  LIN {X -999.998,Y -0.298,Z -43.502,A -90.00011,B 0.00000,C -180.00000} ; release
  LIN {X -999.998,Y -0.298,Z 256.498,A -90.00011,B 0.00000,C -180.00000} ; retreat
  ; Step 2683, bar 145
  LIN {X -874.998,Y -0.298,Z 1164.733,A -90.00011,B 0.00000,C -180.00000} ; outside
  LIN {X -874.998,Y -0.298,Z 206.498,A -90.00011,B 0.00000,C -180.00000} ; preinsert
  LIN {X -874.998,Y -0.298,Z -43.502,A -90.00011,B 0.00000,C -180.00000} ; insert
  LIN {X -874.998,Y -0.298,Z -43.502,A -90.00011,B 0.00000,C -180.00000} ; release
  LIN {X -874.998,Y -0.298,Z 256.498,A -90.00011,B 0.00000,C -180.00000} ; retreat
  ; Step 2684, bar 144
  LIN {X -749.998,Y -0.298,Z 1164.733,A -90.00011,B 0.00000,C -180.00000} ; outside
  LIN {X -749.998,Y -0.298,Z 206.498,A -90.00011,B 0.00000,C -180.00000} ; preinsert
  LIN {X -749.998,Y -0.298,Z -43.502,A -90.00011,B 0.00000,C -180.00000} ; insert
  LIN {X -749.998,Y -0.298,Z -43.502,A -90.00011,B 0.00000,C -180.00000} ; release
  LIN {X -749.998,Y -0.298,Z 256.498,A -90.00011,B 0.00000,C -180.00000} ; retreat
  ; Step 2685, bar 143
  LIN {X -624.998,Y -0.298,Z 1164.733,A -90.00011,B 0.00000,C -180.00000} ; outside
  LIN {X -624.998,Y -0.298,Z 206.498,A -90.00011,B 0.00000,C -180.00000} ; preinsert
  LIN {X -624.998,Y -0.298,Z -43.502,A -90.00011,B 0.00000,C -180.00000} ; insert
  LIN {X -624.998,Y -0.298,Z -43.502,A -90.00011,B 0.00000,C -180.00000} ; release
  LIN {X -624.998,Y -0.298,Z 256.498,A -90.00011,B 0.00000,C -180.00000} ; retreat
  ; Step 2686, bar 142
  LIN {X -499.998,Y -0.298,Z 1164.733,A -90.00011,B 0.00000,C -180.00000} ; outside
  LIN {X -499.998,Y -0.298,Z 206.498,A -90.00011,B 0.00000,C -180.00000} ; preinsert
  LIN {X -499.998,Y -0.298,Z -43.502,A -90.00011,B 0.00000,C -180.00000} ; insert
  LIN {X -499.998,Y -0.298,Z -43.502,A -90.00011,B 0.00000,C -180.00000} ; release
  LIN {X -499.998,Y -0.298,Z 256.498,A -90.00011,B 0.00000,C -180.00000} ; retreat
  ; Step 2687, bar 141
  LIN {X -374.998,Y -0.298,Z 1164.733,A -90.00011,B 0.00000,C -180.00000} ; outside
  LIN {X -374.998,Y -0.298,Z 206.498,A -90.00011,B 0.00000,C -180.00000} ; preinsert
  LIN {X -374.998,Y -0.298,Z -43.502,A -90.00011,B 0.00000,C -180.00000} ; insert
  LIN {X -374.998,Y -0.298,Z -43.502,A -90.00011,B 0.00000,C -180.00000} ; release
  LIN {X -374.998,Y -0.298,Z 256.498,A -90.00011,B 0.00000,C -180.00000} ; retreat
  ; Step 2688, bar 140
  LIN {X -249.998,Y -0.298,Z 1164.733,A -90.00011,B 0.00000,C -180.00000} ; outside
  LIN {X -249.998,Y -0.298,Z 206.498,A -90.00011,B 0.00000,C -180.00000} ; preinsert
  LIN {X -249.998,Y -0.298,Z -43.502,A -90.00011,B 0.00000,C -180.00000} ; insert
  LIN {X -249.998,Y -0.298,Z -43.502,A -90.00011,B 0.00000,C -180.00000} ; release
  LIN {X -249.998,Y -0.298,Z 256.498,A -90.00011,B 0.00000,C -180.00000} ; retreat
  ; Step 2689, bar 139
  LIN {X -124.998,Y -0.298,Z 1164.733,A -90.00011,B 0.00000,C -180.00000} ; outside
  LIN {X -124.998,Y -0.298,Z 206.498,A -90.00011,B 0.00000,C -180.00000} ; preinsert
  LIN {X -124.998,Y -0.298,Z -43.502,A -90.00011,B 0.00000,C -180.00000} ; insert
  LIN {X -124.998,Y -0.298,Z -43.502,A -90.00011,B 0.00000,C -180.00000} ; release
  LIN {X -124.998,Y -0.298,Z 256.498,A -90.00011,B 0.00000,C -180.00000} ; retreat
  ; Step 2690, bar 0
  LIN {X -0.034,Y -0.300,Z 1164.951,A -90.01312,B 0.00000,C -180.00000} ; outside
  LIN {X -0.034,Y -0.300,Z 206.586,A -90.01312,B 0.00000,C -180.00000} ; preinsert
  LIN {X -0.034,Y -0.300,Z -43.414,A -90.01312,B 0.00000,C -180.00000} ; insert
  LIN {X -0.034,Y -0.300,Z -43.414,A -90.01312,B 0.00000,C -180.00000} ; release
  LIN {X -0.034,Y -0.300,Z 256.586,A -90.01312,B 0.00000,C -180.00000} ; retreat
  ; Step 2691, bar 1
  LIN {X 124.966,Y -0.300,Z 1164.951,A -90.01312,B 0.00000,C -180.00000} ; outside
  LIN {X 124.966,Y -0.300,Z 206.586,A -90.01312,B 0.00000,C -180.00000} ; preinsert
  LIN {X 124.966,Y -0.300,Z -43.414,A -90.01312,B 0.00000,C -180.00000} ; insert
  LIN {X 124.966,Y -0.300,Z -43.414,A -90.01312,B 0.00000,C -180.00000} ; release
  LIN {X 124.966,Y -0.300,Z 256.586,A -90.01312,B 0.00000,C -180.00000} ; retreat
  ; Step 2692, bar 2
  LIN {X 249.966,Y -0.300,Z 1164.951,A -90.01312,B 0.00000,C -180.00000} ; outside
  LIN {X 249.966,Y -0.300,Z 206.586,A -90.01312,B 0.00000,C -180.00000} ; preinsert
  LIN {X 249.966,Y -0.300,Z -43.414,A -90.01312,B 0.00000,C -180.00000} ; insert
  LIN {X 249.966,Y -0.300,Z -43.414,A -90.01312,B 0.00000,C -180.00000} ; release
  LIN {X 249.966,Y -0.300,Z 256.586,A -90.01312,B 0.00000,C -180.00000} ; retreat
  ; Step 2693, bar 3
  LIN {X 374.966,Y -0.300,Z 1164.951,A -90.01312,B 0.00000,C -180.00000} ; outside
  LIN {X 374.966,Y -0.300,Z 206.586,A -90.01312,B 0.00000,C -180.00000} ; preinsert
  LIN {X 374.966,Y -0.300,Z -43.414,A -90.01312,B 0.00000,C -180.00000} ; insert
  LIN {X 374.966,Y -0.300,Z -43.414,A -90.01312,B 0.00000,C -180.00000} ; release
  LIN {X 374.966,Y -0.300,Z 256.586,A -90.01312,B 0.00000,C -180.00000} ; retreat
  ; Step 2694, bar 4
  LIN {X 499.966,Y -0.300,Z 1164.951,A -90.01312,B 0.00000,C -180.00000} ; outside
  LIN {X 499.966,Y -0.300,Z 206.586,A -90.01312,B 0.00000,C -180.00000} ; preinsert
  LIN {X 499.966,Y -0.300,Z -43.414,A -90.01312,B 0.00000,C -180.00000} ; insert
  LIN {X 499.966,Y -0.300,Z -43.414,A -90.01312,B 0.00000,C -180.00000} ; release
  LIN {X 499.966,Y -0.300,Z 256.586,A -90.01312,B 0.00000,C -180.00000} ; retreat
  ; Step 2695, bar 5
  LIN {X 624.966,Y -0.300,Z 1164.951,A -90.01312,B 0.00000,C -180.00000} ; outside
  LIN {X 624.966,Y -0.300,Z 206.586,A -90.01312,B 0.00000,C -180.00000} ; preinsert
  LIN {X 624.966,Y -0.300,Z -43.414,A -90.01312,B 0.00000,C -180.00000} ; insert
  LIN {X 624.966,Y -0.300,Z -43.414,A -90.01312,B 0.00000,C -180.00000} ; release
  LIN {X 624.966,Y -0.300,Z 256.586,A -90.01312,B 0.00000,C -180.00000} ; retreat
  ; Step 2696, bar 6
  LIN {X 749.966,Y -0.300,Z 1164.951,A -90.01312,B 0.00000,C -180.00000} ; outside
  LIN {X 749.966,Y -0.300,Z 206.586,A -90.01312,B 0.00000,C -180.00000} ; preinsert
  LIN {X 749.966,Y -0.300,Z -43.414,A -90.01312,B 0.00000,C -180.00000} ; insert
  LIN {X 749.966,Y -0.300,Z -43.414,A -90.01312,B 0.00000,C -180.00000} ; release
  LIN {X 749.966,Y -0.300,Z 256.586,A -90.01312,B 0.00000,C -180.00000} ; retreat
  ; Step 2697, bar 7
  LIN {X 874.966,Y -0.300,Z 1164.951,A -90.01312,B 0.00000,C -180.00000} ; outside
  LIN {X 874.966,Y -0.300,Z 206.586,A -90.01312,B 0.00000,C -180.00000} ; preinsert
  LIN {X 874.966,Y -0.300,Z -43.414,A -90.01312,B 0.00000,C -180.00000} ; insert
  LIN {X 874.966,Y -0.300,Z -43.414,A -90.01312,B 0.00000,C -180.00000} ; release
  LIN {X 874.966,Y -0.300,Z 256.586,A -90.01312,B 0.00000,C -180.00000} ; retreat
  ; Step 2698, bar 8
  LIN {X 999.966,Y -0.300,Z 1164.951,A -90.01312,B 0.00000,C -180.00000} ; outside
  LIN {X 999.966,Y -0.300,Z 206.586,A -90.01312,B 0.00000,C -180.00000} ; preinsert
  LIN {X 999.966,Y -0.300,Z -43.414,A -90.01312,B 0.00000,C -180.00000} ; insert
  LIN {X 999.966,Y -0.300,Z -43.414,A -90.01312,B 0.00000,C -180.00000} ; release
  LIN {X 999.966,Y -0.300,Z 256.586,A -90.01312,B 0.00000,C -180.00000} ; retreat
  ; Step 2699, bar 9
  LIN {X 1124.966,Y -0.300,Z 1164.951,A -90.01312,B 0.00000,C -180.00000} ; outside
  LIN {X 1124.966,Y -0.300,Z 206.586,A -90.01312,B 0.00000,C -180.00000} ; preinsert
  LIN {X 1124.966,Y -0.300,Z -43.414,A -90.01312,B 0.00000,C -180.00000} ; insert
  LIN {X 1124.966,Y -0.300,Z -43.414,A -90.01312,B 0.00000,C -180.00000} ; release
  LIN {X 1124.966,Y -0.300,Z 256.586,A -90.01312,B 0.00000,C -180.00000} ; retreat
  ; Step 2700, bar 10
  LIN {X 1249.966,Y -0.300,Z 1164.951,A -90.01312,B 0.00000,C -180.00000} ; outside
  LIN {X 1249.966,Y -0.300,Z 206.586,A -90.01312,B 0.00000,C -180.00000} ; preinsert
  LIN {X 1249.966,Y -0.300,Z -43.414,A -90.01312,B 0.00000,C -180.00000} ; insert
  LIN {X 1249.966,Y -0.300,Z -43.414,A -90.01312,B 0.00000,C -180.00000} ; release
  LIN {X 1249.966,Y -0.300,Z 256.586,A -90.01312,B 0.00000,C -180.00000} ; retreat
  ; Step 2701, bar 11
  LIN {X 1374.966,Y -0.300,Z 1164.951,A -90.01312,B 0.00000,C -180.00000} ; outside
  LIN {X 1374.966,Y -0.300,Z 206.586,A -90.01312,B 0.00000,C -180.00000} ; preinsert
  LIN {X 1374.966,Y -0.300,Z -43.414,A -90.01312,B 0.00000,C -180.00000} ; insert
  LIN {X 1374.966,Y -0.300,Z -43.414,A -90.01312,B 0.00000,C -180.00000} ; release
  LIN {X 1374.966,Y -0.300,Z 256.586,A -90.01312,B 0.00000,C -180.00000} ; retreat
  ; Step 2702, bar 12
  LIN {X 1499.966,Y -0.300,Z 1164.951,A -90.01312,B 0.00000,C -180.00000} ; outside
  LIN {X 1499.966,Y -0.300,Z 206.586,A -90.01312,B 0.00000,C -180.00000} ; preinsert
  LIN {X 1499.966,Y -0.300,Z -43.414,A -90.01312,B 0.00000,C -180.00000} ; insert
  LIN {X 1499.966,Y -0.300,Z -43.414,A -90.01312,B 0.00000,C -180.00000} ; release
  LIN {X 1499.966,Y -0.300,Z 256.586,A -90.01312,B 0.00000,C -180.00000} ; retreat
  ; Step 2703, bar 13
  LIN {X 1624.966,Y -0.300,Z 1164.951,A -90.01312,B 0.00000,C -180.00000} ; outside
  LIN {X 1624.966,Y -0.300,Z 206.586,A -90.01312,B 0.00000,C -180.00000} ; preinsert
  LIN {X 1624.966,Y -0.300,Z -43.414,A -90.01312,B 0.00000,C -180.00000} ; insert
  LIN {X 1624.966,Y -0.300,Z -43.414,A -90.01312,B 0.00000,C -180.00000} ; release
  LIN {X 1624.966,Y -0.300,Z 256.586,A -90.01312,B 0.00000,C -180.00000} ; retreat
  ; Step 2704, bar 14
  LIN {X 1749.966,Y -0.300,Z 1164.951,A -90.01312,B 0.00000,C -180.00000} ; outside
  LIN {X 1749.966,Y -0.300,Z 206.586,A -90.01312,B 0.00000,C -180.00000} ; preinsert
  LIN {X 1749.966,Y -0.300,Z -43.414,A -90.01312,B 0.00000,C -180.00000} ; insert
  LIN {X 1749.966,Y -0.300,Z -43.414,A -90.01312,B 0.00000,C -180.00000} ; release
  LIN {X 1749.966,Y -0.300,Z 256.586,A -90.01312,B 0.00000,C -180.00000} ; retreat
  ; Step 2705, bar 16
  LIN {X 1874.966,Y -0.300,Z 1164.951,A -90.01312,B 0.00000,C -180.00000} ; outside
  LIN {X 1874.966,Y -0.300,Z 206.586,A -90.01312,B 0.00000,C -180.00000} ; preinsert
  LIN {X 1874.966,Y -0.300,Z -43.414,A -90.01312,B 0.00000,C -180.00000} ; insert
  LIN {X 1874.966,Y -0.300,Z -43.414,A -90.01312,B 0.00000,C -180.00000} ; release
  LIN {X 1874.966,Y -0.300,Z 256.586,A -90.01312,B 0.00000,C -180.00000} ; retreat
  ; Step 2706, bar 17
  LIN {X 2124.966,Y -0.300,Z 1164.951,A -90.01312,B 0.00000,C -180.00000} ; outside
  LIN {X 2124.966,Y -0.300,Z 206.586,A -90.01312,B 0.00000,C -180.00000} ; preinsert
  LIN {X 2124.966,Y -0.300,Z -43.414,A -90.01312,B 0.00000,C -180.00000} ; insert
  LIN {X 2124.966,Y -0.300,Z -43.414,A -90.01312,B 0.00000,C -180.00000} ; release
  LIN {X 2124.966,Y -0.300,Z 256.586,A -90.01312,B 0.00000,C -180.00000} ; retreat
  ; Step 2707, bar 18
  LIN {X 2249.966,Y -0.300,Z 1164.951,A -90.01312,B 0.00000,C -180.00000} ; outside
  LIN {X 2249.966,Y -0.300,Z 206.586,A -90.01312,B 0.00000,C -180.00000} ; preinsert
  LIN {X 2249.966,Y -0.300,Z -43.414,A -90.01312,B 0.00000,C -180.00000} ; insert
  LIN {X 2249.966,Y -0.300,Z -43.414,A -90.01312,B 0.00000,C -180.00000} ; release
  LIN {X 2249.966,Y -0.300,Z 256.586,A -90.01312,B 0.00000,C -180.00000} ; retreat
  ; Step 2708, bar 19
  LIN {X 2374.966,Y -0.300,Z 1164.951,A -90.01312,B 0.00000,C -180.00000} ; outside
  LIN {X 2374.966,Y -0.300,Z 206.586,A -90.01312,B 0.00000,C -180.00000} ; preinsert
  LIN {X 2374.966,Y -0.300,Z -43.414,A -90.01312,B 0.00000,C -180.00000} ; insert
  LIN {X 2374.966,Y -0.300,Z -43.414,A -90.01312,B 0.00000,C -180.00000} ; release
  LIN {X 2374.966,Y -0.300,Z 256.586,A -90.01312,B 0.00000,C -180.00000} ; retreat
  ; Step 2709, bar 20
  LIN {X 2499.966,Y -0.300,Z 1164.951,A -90.01312,B 0.00000,C -180.00000} ; outside
  LIN {X 2499.966,Y -0.300,Z 206.586,A -90.01312,B 0.00000,C -180.00000} ; preinsert
  LIN {X 2499.966,Y -0.300,Z -43.414,A -90.01312,B 0.00000,C -180.00000} ; insert
  LIN {X 2499.966,Y -0.300,Z -43.414,A -90.01312,B 0.00000,C -180.00000} ; release
  LIN {X 2499.966,Y -0.300,Z 256.586,A -90.01312,B 0.00000,C -180.00000} ; retreat
  ; Step 2710, bar 21
  LIN {X 2624.966,Y -0.300,Z 1164.951,A -90.01312,B 0.00000,C -180.00000} ; outside
  LIN {X 2624.966,Y -0.300,Z 206.586,A -90.01312,B 0.00000,C -180.00000} ; preinsert
  LIN {X 2624.966,Y -0.300,Z -43.414,A -90.01312,B 0.00000,C -180.00000} ; insert
  LIN {X 2624.966,Y -0.300,Z -43.414,A -90.01312,B 0.00000,C -180.00000} ; release
  LIN {X 2624.966,Y -0.300,Z 256.586,A -90.01312,B 0.00000,C -180.00000} ; retreat
  ; Step 2711, bar 22
  LIN {X 2749.966,Y -0.300,Z 1164.951,A -90.01312,B 0.00000,C -180.00000} ; outside
  LIN {X 2749.966,Y -0.300,Z 206.586,A -90.01312,B 0.00000,C -180.00000} ; preinsert
  LIN {X 2749.966,Y -0.300,Z -43.414,A -90.01312,B 0.00000,C -180.00000} ; insert
  LIN {X 2749.966,Y -0.300,Z -43.414,A -90.01312,B 0.00000,C -180.00000} ; release
  LIN {X 2749.966,Y -0.300,Z 256.586,A -90.01312,B 0.00000,C -180.00000} ; retreat
  ; Step 2712, bar 23
  LIN {X 2874.966,Y -0.300,Z 1164.951,A -90.01312,B 0.00000,C -180.00000} ; outside
  LIN {X 2874.966,Y -0.300,Z 206.586,A -90.01312,B 0.00000,C -180.00000} ; preinsert
  LIN {X 2874.966,Y -0.300,Z -43.414,A -90.01312,B 0.00000,C -180.00000} ; insert
  LIN {X 2874.966,Y -0.300,Z -43.414,A -90.01312,B 0.00000,C -180.00000} ; release
  LIN {X 2874.966,Y -0.300,Z 256.586,A -90.01312,B 0.00000,C -180.00000} ; retreat
  ; Step 2713, bar 24
  LIN {X 2999.966,Y -0.300,Z 1164.951,A -90.01312,B 0.00000,C -180.00000} ; outside
  LIN {X 2999.966,Y -0.300,Z 206.586,A -90.01312,B 0.00000,C -180.00000} ; preinsert
  LIN {X 2999.966,Y -0.300,Z -43.414,A -90.01312,B 0.00000,C -180.00000} ; insert
  LIN {X 2999.966,Y -0.300,Z -43.414,A -90.01312,B 0.00000,C -180.00000} ; release
  LIN {X 2999.966,Y -0.300,Z 256.586,A -90.01312,B 0.00000,C -180.00000} ; retreat
  ; Step 2714, bar 25
  LIN {X 3124.966,Y -0.300,Z 1164.951,A -90.01312,B 0.00000,C -180.00000} ; outside
  LIN {X 3124.966,Y -0.300,Z 206.586,A -90.01312,B 0.00000,C -180.00000} ; preinsert
  LIN {X 3124.966,Y -0.300,Z -43.414,A -90.01312,B 0.00000,C -180.00000} ; insert
  LIN {X 3124.966,Y -0.300,Z -43.414,A -90.01312,B 0.00000,C -180.00000} ; release
  LIN {X 3124.966,Y -0.300,Z 256.586,A -90.01312,B 0.00000,C -180.00000} ; retreat
  ; Step 2715, bar 26
  LIN {X 3249.966,Y -0.300,Z 1164.951,A -90.01312,B 0.00000,C -180.00000} ; outside
  LIN {X 3249.966,Y -0.300,Z 206.586,A -90.01312,B 0.00000,C -180.00000} ; preinsert
  LIN {X 3249.966,Y -0.300,Z -43.414,A -90.01312,B 0.00000,C -180.00000} ; insert
  LIN {X 3249.966,Y -0.300,Z -43.414,A -90.01312,B 0.00000,C -180.00000} ; release
  LIN {X 3249.966,Y -0.300,Z 256.586,A -90.01312,B 0.00000,C -180.00000} ; retreat
  ; Step 2716, bar 27
  LIN {X 3374.966,Y -0.300,Z 1164.951,A -90.01312,B 0.00000,C -180.00000} ; outside
  LIN {X 3374.966,Y -0.300,Z 206.586,A -90.01312,B 0.00000,C -180.00000} ; preinsert
  LIN {X 3374.966,Y -0.300,Z -43.414,A -90.01312,B 0.00000,C -180.00000} ; insert
  LIN {X 3374.966,Y -0.300,Z -43.414,A -90.01312,B 0.00000,C -180.00000} ; release
  LIN {X 3374.966,Y -0.300,Z 256.586,A -90.01312,B 0.00000,C -180.00000} ; retreat
  ; Step 2717, bar 28
  LIN {X 3499.966,Y -0.300,Z 1164.951,A -90.01312,B 0.00000,C -180.00000} ; outside
  LIN {X 3499.966,Y -0.300,Z 206.586,A -90.01312,B 0.00000,C -180.00000} ; preinsert
  LIN {X 3499.966,Y -0.300,Z -43.414,A -90.01312,B 0.00000,C -180.00000} ; insert
  LIN {X 3499.966,Y -0.300,Z -43.414,A -90.01312,B 0.00000,C -180.00000} ; release
  LIN {X 3499.966,Y -0.300,Z 256.586,A -90.01312,B 0.00000,C -180.00000} ; retreat
  ; Step 2718, bar 29
  LIN {X 3624.966,Y -0.300,Z 1164.951,A -90.01312,B 0.00000,C -180.00000} ; outside
  LIN {X 3624.966,Y -0.300,Z 206.586,A -90.01312,B 0.00000,C -180.00000} ; preinsert
  LIN {X 3624.966,Y -0.300,Z -43.414,A -90.01312,B 0.00000,C -180.00000} ; insert
  LIN {X 3624.966,Y -0.300,Z -43.414,A -90.01312,B 0.00000,C -180.00000} ; release
  LIN {X 3624.966,Y -0.300,Z 256.586,A -90.01312,B 0.00000,C -180.00000} ; retreat
  ; Step 2719, bar 30
  LIN {X 3749.966,Y -0.300,Z 1164.951,A -90.01312,B 0.00000,C -180.00000} ; outside
  LIN {X 3749.966,Y -0.300,Z 206.586,A -90.01312,B 0.00000,C -180.00000} ; preinsert
  LIN {X 3749.966,Y -0.300,Z -43.414,A -90.01312,B 0.00000,C -180.00000} ; insert
  LIN {X 3749.966,Y -0.300,Z -43.414,A -90.01312,B 0.00000,C -180.00000} ; release
  LIN {X 3749.966,Y -0.300,Z 256.586,A -90.01312,B 0.00000,C -180.00000} ; retreat
  ; Step 2720, bar 31
  LIN {X 3874.966,Y -0.300,Z 1164.951,A -90.01312,B 0.00000,C -180.00000} ; outside
  LIN {X 3874.966,Y -0.300,Z 206.586,A -90.01312,B 0.00000,C -180.00000} ; preinsert
  LIN {X 3874.966,Y -0.300,Z -43.414,A -90.01312,B 0.00000,C -180.00000} ; insert
  LIN {X 3874.966,Y -0.300,Z -43.414,A -90.01312,B 0.00000,C -180.00000} ; release
  LIN {X 3874.966,Y -0.300,Z 256.586,A -90.01312,B 0.00000,C -180.00000} ; retreat
  ; Step 2721, bar 32
  LIN {X 3999.966,Y -0.300,Z 1164.951,A -90.01312,B 0.00000,C -180.00000} ; outside
  LIN {X 3999.966,Y -0.300,Z 206.586,A -90.01312,B 0.00000,C -180.00000} ; preinsert
  LIN {X 3999.966,Y -0.300,Z -43.414,A -90.01312,B 0.00000,C -180.00000} ; insert
  LIN {X 3999.966,Y -0.300,Z -43.414,A -90.01312,B 0.00000,C -180.00000} ; release
  LIN {X 3999.966,Y -0.300,Z 256.586,A -90.01312,B 0.00000,C -180.00000} ; retreat
  ; Step 2722, bar 33
  LIN {X 4124.966,Y -0.300,Z 1164.951,A -90.01312,B 0.00000,C -180.00000} ; outside
  LIN {X 4124.966,Y -0.300,Z 206.586,A -90.01312,B 0.00000,C -180.00000} ; preinsert
  LIN {X 4124.966,Y -0.300,Z -43.414,A -90.01312,B 0.00000,C -180.00000} ; insert
  LIN {X 4124.966,Y -0.300,Z -43.414,A -90.01312,B 0.00000,C -180.00000} ; release
  LIN {X 4124.966,Y -0.300,Z 256.586,A -90.01312,B 0.00000,C -180.00000} ; retreat
  ; Step 2723, bar 34
  LIN {X 4249.966,Y -0.300,Z 1164.951,A -90.01312,B 0.00000,C -180.00000} ; outside
  LIN {X 4249.966,Y -0.300,Z 206.586,A -90.01312,B 0.00000,C -180.00000} ; preinsert
  LIN {X 4249.966,Y -0.300,Z -43.414,A -90.01312,B 0.00000,C -180.00000} ; insert
  LIN {X 4249.966,Y -0.300,Z -43.414,A -90.01312,B 0.00000,C -180.00000} ; release
  LIN {X 4249.966,Y -0.300,Z 256.586,A -90.01312,B 0.00000,C -180.00000} ; retreat
  ; Step 2724, bar 35
  LIN {X 4374.966,Y -0.300,Z 1164.951,A -90.01312,B 0.00000,C -180.00000} ; outside
  LIN {X 4374.966,Y -0.300,Z 206.586,A -90.01312,B 0.00000,C -180.00000} ; preinsert
  LIN {X 4374.966,Y -0.300,Z -43.414,A -90.01312,B 0.00000,C -180.00000} ; insert
  LIN {X 4374.966,Y -0.300,Z -43.414,A -90.01312,B 0.00000,C -180.00000} ; release
  LIN {X 4374.966,Y -0.300,Z 256.586,A -90.01312,B 0.00000,C -180.00000} ; retreat
  ; Step 2725, bar 36
  LIN {X 4499.966,Y -0.300,Z 1164.951,A -90.01312,B 0.00000,C -180.00000} ; outside
  LIN {X 4499.966,Y -0.300,Z 206.586,A -90.01312,B 0.00000,C -180.00000} ; preinsert
  LIN {X 4499.966,Y -0.300,Z -43.414,A -90.01312,B 0.00000,C -180.00000} ; insert
  LIN {X 4499.966,Y -0.300,Z -43.414,A -90.01312,B 0.00000,C -180.00000} ; release
  LIN {X 4499.966,Y -0.300,Z 256.586,A -90.01312,B 0.00000,C -180.00000} ; retreat
  ; Step 2726, bar 37
  LIN {X 4624.966,Y -0.300,Z 1164.951,A -90.01312,B 0.00000,C -180.00000} ; outside
  LIN {X 4624.966,Y -0.300,Z 206.586,A -90.01312,B 0.00000,C -180.00000} ; preinsert
  LIN {X 4624.966,Y -0.300,Z -43.414,A -90.01312,B 0.00000,C -180.00000} ; insert
  LIN {X 4624.966,Y -0.300,Z -43.414,A -90.01312,B 0.00000,C -180.00000} ; release
  LIN {X 4624.966,Y -0.300,Z 256.586,A -90.01312,B 0.00000,C -180.00000} ; retreat
  ; Step 2727, bar 38
  LIN {X 4749.966,Y -0.300,Z 1164.951,A -90.01312,B 0.00000,C -180.00000} ; outside
  LIN {X 4749.966,Y -0.300,Z 206.586,A -90.01312,B 0.00000,C -180.00000} ; preinsert
  LIN {X 4749.966,Y -0.300,Z -43.414,A -90.01312,B 0.00000,C -180.00000} ; insert
  LIN {X 4749.966,Y -0.300,Z -43.414,A -90.01312,B 0.00000,C -180.00000} ; release
  LIN {X 4749.966,Y -0.300,Z 256.586,A -90.01312,B 0.00000,C -180.00000} ; retreat
  ; Step 2728, bar 39
  LIN {X 4874.966,Y -0.300,Z 1164.951,A -90.01312,B 0.00000,C -180.00000} ; outside
  LIN {X 4874.966,Y -0.300,Z 206.586,A -90.01312,B 0.00000,C -180.00000} ; preinsert
  LIN {X 4874.966,Y -0.300,Z -43.414,A -90.01312,B 0.00000,C -180.00000} ; insert
  LIN {X 4874.966,Y -0.300,Z -43.414,A -90.01312,B 0.00000,C -180.00000} ; release
  LIN {X 4874.966,Y -0.300,Z 256.586,A -90.01312,B 0.00000,C -180.00000} ; retreat
  ; Step 2729, bar 40
  LIN {X 4999.966,Y -0.300,Z 1164.951,A -90.01312,B 0.00000,C -180.00000} ; outside
  LIN {X 4999.966,Y -0.300,Z 206.586,A -90.01312,B 0.00000,C -180.00000} ; preinsert
  LIN {X 4999.966,Y -0.300,Z -43.414,A -90.01312,B 0.00000,C -180.00000} ; insert
  LIN {X 4999.966,Y -0.300,Z -43.414,A -90.01312,B 0.00000,C -180.00000} ; release
  LIN {X 4999.966,Y -0.300,Z 256.586,A -90.01312,B 0.00000,C -180.00000} ; retreat
  ; Step 2730, bar 41
  LIN {X 5124.966,Y -0.300,Z 1164.951,A -90.01312,B 0.00000,C -180.00000} ; outside
  LIN {X 5124.966,Y -0.300,Z 206.586,A -90.01312,B 0.00000,C -180.00000} ; preinsert
  LIN {X 5124.966,Y -0.300,Z -43.414,A -90.01312,B 0.00000,C -180.00000} ; insert
  LIN {X 5124.966,Y -0.300,Z -43.414,A -90.01312,B 0.00000,C -180.00000} ; release
  LIN {X 5124.966,Y -0.300,Z 256.586,A -90.01312,B 0.00000,C -180.00000} ; retreat
  ; Step 2731, bar 42
  LIN {X 5249.966,Y -0.300,Z 1164.951,A -90.01312,B 0.00000,C -180.00000} ; outside
  LIN {X 5249.966,Y -0.300,Z 206.586,A -90.01312,B 0.00000,C -180.00000} ; preinsert
  LIN {X 5249.966,Y -0.300,Z -43.414,A -90.01312,B 0.00000,C -180.00000} ; insert
  LIN {X 5249.966,Y -0.300,Z -43.414,A -90.01312,B 0.00000,C -180.00000} ; release
  LIN {X 5249.966,Y -0.300,Z 256.586,A -90.01312,B 0.00000,C -180.00000} ; retreat
  ; Step 2732, bar 43
  LIN {X 5374.966,Y -0.300,Z 1164.951,A -90.01312,B 0.00000,C -180.00000} ; outside
  LIN {X 5374.966,Y -0.300,Z 206.586,A -90.01312,B 0.00000,C -180.00000} ; preinsert
  LIN {X 5374.966,Y -0.300,Z -43.414,A -90.01312,B 0.00000,C -180.00000} ; insert
  LIN {X 5374.966,Y -0.300,Z -43.414,A -90.01312,B 0.00000,C -180.00000} ; release
  LIN {X 5374.966,Y -0.300,Z 256.586,A -90.01312,B 0.00000,C -180.00000} ; retreat
  ; Step 2733, bar 44
  LIN {X 5499.966,Y -0.300,Z 1164.951,A -90.01312,B 0.00000,C -180.00000} ; outside
  LIN {X 5499.966,Y -0.300,Z 206.586,A -90.01312,B 0.00000,C -180.00000} ; preinsert
  LIN {X 5499.966,Y -0.300,Z -43.414,A -90.01312,B 0.00000,C -180.00000} ; insert
  LIN {X 5499.966,Y -0.300,Z -43.414,A -90.01312,B 0.00000,C -180.00000} ; release
  LIN {X 5499.966,Y -0.300,Z 256.586,A -90.01312,B 0.00000,C -180.00000} ; retreat
  ; Step 2734, bar 45
  LIN {X 5624.966,Y -0.300,Z 1164.951,A -90.01312,B 0.00000,C -180.00000} ; outside
  LIN {X 5624.966,Y -0.300,Z 206.586,A -90.01312,B 0.00000,C -180.00000} ; preinsert
  LIN {X 5624.966,Y -0.300,Z -43.414,A -90.01312,B 0.00000,C -180.00000} ; insert
  LIN {X 5624.966,Y -0.300,Z -43.414,A -90.01312,B 0.00000,C -180.00000} ; release
  LIN {X 5624.966,Y -0.300,Z 256.586,A -90.01312,B 0.00000,C -180.00000} ; retreat
  ; Step 2735, bar 46
  LIN {X 5749.966,Y -0.300,Z 1164.951,A -90.01312,B 0.00000,C -180.00000} ; outside
  LIN {X 5749.966,Y -0.300,Z 206.586,A -90.01312,B 0.00000,C -180.00000} ; preinsert
  LIN {X 5749.966,Y -0.300,Z -43.414,A -90.01312,B 0.00000,C -180.00000} ; insert
  LIN {X 5749.966,Y -0.300,Z -43.414,A -90.01312,B 0.00000,C -180.00000} ; release
  LIN {X 5749.966,Y -0.300,Z 256.586,A -90.01312,B 0.00000,C -180.00000} ; retreat
  ; Step 2736, bar 48
  LIN {X 5874.966,Y -0.300,Z 1164.951,A -90.01312,B 0.00000,C -180.00000} ; outside
  LIN {X 5874.966,Y -0.300,Z 206.586,A -90.01312,B 0.00000,C -180.00000} ; preinsert
  LIN {X 5874.966,Y -0.300,Z -43.414,A -90.01312,B 0.00000,C -180.00000} ; insert
  LIN {X 5874.966,Y -0.300,Z -43.414,A -90.01312,B 0.00000,C -180.00000} ; release
  LIN {X 5874.966,Y -0.300,Z 256.586,A -90.01312,B 0.00000,C -180.00000} ; retreat
  ; Step 2737, bar 49
  LIN {X 6124.966,Y -0.300,Z 1164.951,A -90.01312,B 0.00000,C -180.00000} ; outside
  LIN {X 6124.966,Y -0.300,Z 206.586,A -90.01312,B 0.00000,C -180.00000} ; preinsert
  LIN {X 6124.966,Y -0.300,Z -43.414,A -90.01312,B 0.00000,C -180.00000} ; insert
  LIN {X 6124.966,Y -0.300,Z -43.414,A -90.01312,B 0.00000,C -180.00000} ; release
  LIN {X 6124.966,Y -0.300,Z 256.586,A -90.01312,B 0.00000,C -180.00000} ; retreat
  ; Step 2738, bar 50
  LIN {X 6249.966,Y -0.300,Z 1164.951,A -90.01312,B 0.00000,C -180.00000} ; outside
  LIN {X 6249.966,Y -0.300,Z 206.586,A -90.01312,B 0.00000,C -180.00000} ; preinsert
  LIN {X 6249.966,Y -0.300,Z -43.414,A -90.01312,B 0.00000,C -180.00000} ; insert
  LIN {X 6249.966,Y -0.300,Z -43.414,A -90.01312,B 0.00000,C -180.00000} ; release
  LIN {X 6249.966,Y -0.300,Z 256.586,A -90.01312,B 0.00000,C -180.00000} ; retreat
  ; Step 2739, bar 51
  LIN {X 6374.966,Y -0.300,Z 1164.951,A -90.01312,B 0.00000,C -180.00000} ; outside
  LIN {X 6374.966,Y -0.300,Z 206.586,A -90.01312,B 0.00000,C -180.00000} ; preinsert
  LIN {X 6374.966,Y -0.300,Z -43.414,A -90.01312,B 0.00000,C -180.00000} ; insert
  LIN {X 6374.966,Y -0.300,Z -43.414,A -90.01312,B 0.00000,C -180.00000} ; release
  LIN {X 6374.966,Y -0.300,Z 256.586,A -90.01312,B 0.00000,C -180.00000} ; retreat
  ; Step 2740, bar 52
  LIN {X 6499.966,Y -0.300,Z 1164.951,A -90.01312,B 0.00000,C -180.00000} ; outside
  LIN {X 6499.966,Y -0.300,Z 206.586,A -90.01312,B 0.00000,C -180.00000} ; preinsert
  LIN {X 6499.966,Y -0.300,Z -43.414,A -90.01312,B 0.00000,C -180.00000} ; insert
  LIN {X 6499.966,Y -0.300,Z -43.414,A -90.01312,B 0.00000,C -180.00000} ; release
  LIN {X 6499.966,Y -0.300,Z 256.586,A -90.01312,B 0.00000,C -180.00000} ; retreat
  ; Step 2741, bar 53
  LIN {X 6624.966,Y -0.300,Z 1164.951,A -90.01312,B 0.00000,C -180.00000} ; outside
  LIN {X 6624.966,Y -0.300,Z 206.586,A -90.01312,B 0.00000,C -180.00000} ; preinsert
  LIN {X 6624.966,Y -0.300,Z -43.414,A -90.01312,B 0.00000,C -180.00000} ; insert
  LIN {X 6624.966,Y -0.300,Z -43.414,A -90.01312,B 0.00000,C -180.00000} ; release
  LIN {X 6624.966,Y -0.300,Z 256.586,A -90.01312,B 0.00000,C -180.00000} ; retreat
  ; Step 2742, bar 54
  LIN {X 6749.966,Y -0.300,Z 1164.951,A -90.01312,B 0.00000,C -180.00000} ; outside
  LIN {X 6749.966,Y -0.300,Z 206.586,A -90.01312,B 0.00000,C -180.00000} ; preinsert
  LIN {X 6749.966,Y -0.300,Z -43.414,A -90.01312,B 0.00000,C -180.00000} ; insert
  LIN {X 6749.966,Y -0.300,Z -43.414,A -90.01312,B 0.00000,C -180.00000} ; release
  LIN {X 6749.966,Y -0.300,Z 256.586,A -90.01312,B 0.00000,C -180.00000} ; retreat
  ; Step 2743, bar 55
  LIN {X 6874.966,Y -0.300,Z 1164.951,A -90.01312,B 0.00000,C -180.00000} ; outside
  LIN {X 6874.966,Y -0.300,Z 206.586,A -90.01312,B 0.00000,C -180.00000} ; preinsert
  LIN {X 6874.966,Y -0.300,Z -43.414,A -90.01312,B 0.00000,C -180.00000} ; insert
  LIN {X 6874.966,Y -0.300,Z -43.414,A -90.01312,B 0.00000,C -180.00000} ; release
  LIN {X 6874.966,Y -0.300,Z 256.586,A -90.01312,B 0.00000,C -180.00000} ; retreat
  ; Step 2744, bar 56
  LIN {X 6999.966,Y -0.300,Z 1164.951,A -90.01312,B 0.00000,C -180.00000} ; outside
  LIN {X 6999.966,Y -0.300,Z 206.586,A -90.01312,B 0.00000,C -180.00000} ; preinsert
  LIN {X 6999.966,Y -0.300,Z -43.414,A -90.01312,B 0.00000,C -180.00000} ; insert
  LIN {X 6999.966,Y -0.300,Z -43.414,A -90.01312,B 0.00000,C -180.00000} ; release
  LIN {X 6999.966,Y -0.300,Z 256.586,A -90.01312,B 0.00000,C -180.00000} ; retreat
  ; Step 2745, bar 57
  LIN {X 7124.966,Y -0.300,Z 1164.951,A -90.01312,B 0.00000,C -180.00000} ; outside
  LIN {X 7124.966,Y -0.300,Z 206.586,A -90.01312,B 0.00000,C -180.00000} ; preinsert
  LIN {X 7124.966,Y -0.300,Z -43.414,A -90.01312,B 0.00000,C -180.00000} ; insert
  LIN {X 7124.966,Y -0.300,Z -43.414,A -90.01312,B 0.00000,C -180.00000} ; release
  LIN {X 7124.966,Y -0.300,Z 256.586,A -90.01312,B 0.00000,C -180.00000} ; retreat
  ; Step 2746, bar 58
  LIN {X 7249.966,Y -0.300,Z 1164.951,A -90.01312,B 0.00000,C -180.00000} ; outside
  LIN {X 7249.966,Y -0.300,Z 206.586,A -90.01312,B 0.00000,C -180.00000} ; preinsert
  LIN {X 7249.966,Y -0.300,Z -43.414,A -90.01312,B 0.00000,C -180.00000} ; insert
  LIN {X 7249.966,Y -0.300,Z -43.414,A -90.01312,B 0.00000,C -180.00000} ; release
  LIN {X 7249.966,Y -0.300,Z 256.586,A -90.01312,B 0.00000,C -180.00000} ; retreat
  ; Step 2747, bar 59
  LIN {X 7374.966,Y -0.300,Z 1164.951,A -90.01312,B 0.00000,C -180.00000} ; outside
  LIN {X 7374.966,Y -0.300,Z 206.586,A -90.01312,B 0.00000,C -180.00000} ; preinsert
  LIN {X 7374.966,Y -0.300,Z -43.414,A -90.01312,B 0.00000,C -180.00000} ; insert
  LIN {X 7374.966,Y -0.300,Z -43.414,A -90.01312,B 0.00000,C -180.00000} ; release
  LIN {X 7374.966,Y -0.300,Z 256.586,A -90.01312,B 0.00000,C -180.00000} ; retreat
  ; Step 2748, bar 60
  LIN {X 7499.966,Y -0.300,Z 1164.951,A -90.01312,B 0.00000,C -180.00000} ; outside
  LIN {X 7499.966,Y -0.300,Z 206.586,A -90.01312,B 0.00000,C -180.00000} ; preinsert
  LIN {X 7499.966,Y -0.300,Z -43.414,A -90.01312,B 0.00000,C -180.00000} ; insert
  LIN {X 7499.966,Y -0.300,Z -43.414,A -90.01312,B 0.00000,C -180.00000} ; release
  LIN {X 7499.966,Y -0.300,Z 256.586,A -90.01312,B 0.00000,C -180.00000} ; retreat
  ; Step 2749, bar 61
  LIN {X 7624.966,Y -0.300,Z 1164.951,A -90.01312,B 0.00000,C -180.00000} ; outside
  LIN {X 7624.966,Y -0.300,Z 206.586,A -90.01312,B 0.00000,C -180.00000} ; preinsert
  LIN {X 7624.966,Y -0.300,Z -43.414,A -90.01312,B 0.00000,C -180.00000} ; insert
  LIN {X 7624.966,Y -0.300,Z -43.414,A -90.01312,B 0.00000,C -180.00000} ; release
  LIN {X 7624.966,Y -0.300,Z 256.586,A -90.01312,B 0.00000,C -180.00000} ; retreat
  ; Step 2750, bar 62
  LIN {X 7749.966,Y -0.300,Z 1164.951,A -90.01312,B 0.00000,C -180.00000} ; outside
  LIN {X 7749.966,Y -0.300,Z 206.586,A -90.01312,B 0.00000,C -180.00000} ; preinsert
  LIN {X 7749.966,Y -0.300,Z -43.414,A -90.01312,B 0.00000,C -180.00000} ; insert
  LIN {X 7749.966,Y -0.300,Z -43.414,A -90.01312,B 0.00000,C -180.00000} ; release
  LIN {X 7749.966,Y -0.300,Z 256.586,A -90.01312,B 0.00000,C -180.00000} ; retreat
  ; Step 2751, bar 63
  LIN {X 7874.966,Y -0.300,Z 1164.951,A -90.01312,B 0.00000,C -180.00000} ; outside
  LIN {X 7874.966,Y -0.300,Z 206.586,A -90.01312,B 0.00000,C -180.00000} ; preinsert
  LIN {X 7874.966,Y -0.300,Z -43.414,A -90.01312,B 0.00000,C -180.00000} ; insert
  LIN {X 7874.966,Y -0.300,Z -43.414,A -90.01312,B 0.00000,C -180.00000} ; release
  LIN {X 7874.966,Y -0.300,Z 256.586,A -90.01312,B 0.00000,C -180.00000} ; retreat
  ; Step 2752, bar 64
  LIN {X 7999.966,Y -0.300,Z 1164.951,A -90.01312,B 0.00000,C -180.00000} ; outside
  LIN {X 7999.966,Y -0.300,Z 206.586,A -90.01312,B 0.00000,C -180.00000} ; preinsert
  LIN {X 7999.966,Y -0.300,Z -43.414,A -90.01312,B 0.00000,C -180.00000} ; insert
  LIN {X 7999.966,Y -0.300,Z -43.414,A -90.01312,B 0.00000,C -180.00000} ; release
  LIN {X 7999.966,Y -0.300,Z 256.586,A -90.01312,B 0.00000,C -180.00000} ; retreat
  ; Step 2753, bar 65
  LIN {X 8124.966,Y -0.300,Z 1164.951,A -90.01312,B 0.00000,C -180.00000} ; outside
  LIN {X 8124.966,Y -0.300,Z 206.586,A -90.01312,B 0.00000,C -180.00000} ; preinsert
  LIN {X 8124.966,Y -0.300,Z -43.414,A -90.01312,B 0.00000,C -180.00000} ; insert
  LIN {X 8124.966,Y -0.300,Z -43.414,A -90.01312,B 0.00000,C -180.00000} ; release
  LIN {X 8124.966,Y -0.300,Z 256.586,A -90.01312,B 0.00000,C -180.00000} ; retreat
  ; Step 2754, bar 66
  LIN {X 8249.966,Y -0.300,Z 1164.951,A -90.01312,B 0.00000,C -180.00000} ; outside
  LIN {X 8249.966,Y -0.300,Z 206.586,A -90.01312,B 0.00000,C -180.00000} ; preinsert
  LIN {X 8249.966,Y -0.300,Z -43.414,A -90.01312,B 0.00000,C -180.00000} ; insert
  LIN {X 8249.966,Y -0.300,Z -43.414,A -90.01312,B 0.00000,C -180.00000} ; release
  LIN {X 8249.966,Y -0.300,Z 256.586,A -90.01312,B 0.00000,C -180.00000} ; retreat
  ; Step 2755, bar 67
  LIN {X 8374.966,Y -0.300,Z 1164.951,A -90.01312,B 0.00000,C -180.00000} ; outside
  LIN {X 8374.966,Y -0.300,Z 206.586,A -90.01312,B 0.00000,C -180.00000} ; preinsert
  LIN {X 8374.966,Y -0.300,Z -43.414,A -90.01312,B 0.00000,C -180.00000} ; insert
  LIN {X 8374.966,Y -0.300,Z -43.414,A -90.01312,B 0.00000,C -180.00000} ; release
  LIN {X 8374.966,Y -0.300,Z 256.586,A -90.01312,B 0.00000,C -180.00000} ; retreat
  ; Step 2756, bar 68
  LIN {X 8499.966,Y -0.300,Z 1164.951,A -90.01312,B 0.00000,C -180.00000} ; outside
  LIN {X 8499.966,Y -0.300,Z 206.586,A -90.01312,B 0.00000,C -180.00000} ; preinsert
  LIN {X 8499.966,Y -0.300,Z -43.414,A -90.01312,B 0.00000,C -180.00000} ; insert
  LIN {X 8499.966,Y -0.300,Z -43.414,A -90.01312,B 0.00000,C -180.00000} ; release
  LIN {X 8499.966,Y -0.300,Z 256.586,A -90.01312,B 0.00000,C -180.00000} ; retreat
  ; Step 2757, bar 69
  LIN {X 8624.966,Y -0.300,Z 1164.951,A -90.01312,B 0.00000,C -180.00000} ; outside
  LIN {X 8624.966,Y -0.300,Z 206.586,A -90.01312,B 0.00000,C -180.00000} ; preinsert
  LIN {X 8624.966,Y -0.300,Z -43.414,A -90.01312,B 0.00000,C -180.00000} ; insert
  LIN {X 8624.966,Y -0.300,Z -43.414,A -90.01312,B 0.00000,C -180.00000} ; release
  LIN {X 8624.966,Y -0.300,Z 256.586,A -90.01312,B 0.00000,C -180.00000} ; retreat
  ; Step 2758, bar 70
  LIN {X 8749.966,Y -0.300,Z 1164.951,A -90.01312,B 0.00000,C -180.00000} ; outside
  LIN {X 8749.966,Y -0.300,Z 206.586,A -90.01312,B 0.00000,C -180.00000} ; preinsert
  LIN {X 8749.966,Y -0.300,Z -43.414,A -90.01312,B 0.00000,C -180.00000} ; insert
  LIN {X 8749.966,Y -0.300,Z -43.414,A -90.01312,B 0.00000,C -180.00000} ; release
  LIN {X 8749.966,Y -0.300,Z 256.586,A -90.01312,B 0.00000,C -180.00000} ; retreat
  ; Step 2759, bar 71
  LIN {X 8874.966,Y -0.300,Z 1164.951,A -90.01312,B 0.00000,C -180.00000} ; outside
  LIN {X 8874.966,Y -0.300,Z 206.586,A -90.01312,B 0.00000,C -180.00000} ; preinsert
  LIN {X 8874.966,Y -0.300,Z -43.414,A -90.01312,B 0.00000,C -180.00000} ; insert
  LIN {X 8874.966,Y -0.300,Z -43.414,A -90.01312,B 0.00000,C -180.00000} ; release
  LIN {X 8874.966,Y -0.300,Z 256.586,A -90.01312,B 0.00000,C -180.00000} ; retreat
  ; Step 2760, bar 72
  LIN {X 8999.966,Y -0.300,Z 1164.951,A -90.01312,B 0.00000,C -180.00000} ; outside
  LIN {X 8999.966,Y -0.300,Z 206.586,A -90.01312,B 0.00000,C -180.00000} ; preinsert
  LIN {X 8999.966,Y -0.300,Z -43.414,A -90.01312,B 0.00000,C -180.00000} ; insert
  LIN {X 8999.966,Y -0.300,Z -43.414,A -90.01312,B 0.00000,C -180.00000} ; release
  LIN {X 8999.966,Y -0.300,Z 256.586,A -90.01312,B 0.00000,C -180.00000} ; retreat
  ; Step 2761, bar 73
  LIN {X 9124.966,Y -0.300,Z 1164.951,A -90.01312,B 0.00000,C -180.00000} ; outside
  LIN {X 9124.966,Y -0.300,Z 206.586,A -90.01312,B 0.00000,C -180.00000} ; preinsert
  LIN {X 9124.966,Y -0.300,Z -43.414,A -90.01312,B 0.00000,C -180.00000} ; insert
  LIN {X 9124.966,Y -0.300,Z -43.414,A -90.01312,B 0.00000,C -180.00000} ; release
  LIN {X 9124.966,Y -0.300,Z 256.586,A -90.01312,B 0.00000,C -180.00000} ; retreat
  ; Step 2762, bar 74
  LIN {X 9249.966,Y -0.300,Z 1164.951,A -90.01312,B 0.00000,C -180.00000} ; outside
  LIN {X 9249.966,Y -0.300,Z 206.586,A -90.01312,B 0.00000,C -180.00000} ; preinsert
  LIN {X 9249.966,Y -0.300,Z -43.414,A -90.01312,B 0.00000,C -180.00000} ; insert
  LIN {X 9249.966,Y -0.300,Z -43.414,A -90.01312,B 0.00000,C -180.00000} ; release
  LIN {X 9249.966,Y -0.300,Z 256.586,A -90.01312,B 0.00000,C -180.00000} ; retreat
  ; Step 2763, bar 75
  LIN {X 9374.966,Y -0.300,Z 1164.951,A -90.01312,B 0.00000,C -180.00000} ; outside
  LIN {X 9374.966,Y -0.300,Z 206.586,A -90.01312,B 0.00000,C -180.00000} ; preinsert
  LIN {X 9374.966,Y -0.300,Z -43.414,A -90.01312,B 0.00000,C -180.00000} ; insert
  LIN {X 9374.966,Y -0.300,Z -43.414,A -90.01312,B 0.00000,C -180.00000} ; release
  LIN {X 9374.966,Y -0.300,Z 256.586,A -90.01312,B 0.00000,C -180.00000} ; retreat
  ; Step 2764, bar 76
  LIN {X 9499.966,Y -0.300,Z 1164.951,A -90.01312,B 0.00000,C -180.00000} ; outside
  LIN {X 9499.966,Y -0.300,Z 206.586,A -90.01312,B 0.00000,C -180.00000} ; preinsert
  LIN {X 9499.966,Y -0.300,Z -43.414,A -90.01312,B 0.00000,C -180.00000} ; insert
  LIN {X 9499.966,Y -0.300,Z -43.414,A -90.01312,B 0.00000,C -180.00000} ; release
  LIN {X 9499.966,Y -0.300,Z 256.586,A -90.01312,B 0.00000,C -180.00000} ; retreat
  ; Step 2765, bar 77
  LIN {X 9624.966,Y -0.300,Z 1164.951,A -90.01312,B 0.00000,C -180.00000} ; outside
  LIN {X 9624.966,Y -0.300,Z 206.586,A -90.01312,B 0.00000,C -180.00000} ; preinsert
  LIN {X 9624.966,Y -0.300,Z -43.414,A -90.01312,B 0.00000,C -180.00000} ; insert
  LIN {X 9624.966,Y -0.300,Z -43.414,A -90.01312,B 0.00000,C -180.00000} ; release
  LIN {X 9624.966,Y -0.300,Z 256.586,A -90.01312,B 0.00000,C -180.00000} ; retreat
  ; Step 2766, bar 78
  LIN {X 9749.966,Y -0.300,Z 1164.951,A -90.01312,B 0.00000,C -180.00000} ; outside
  LIN {X 9749.966,Y -0.300,Z 206.586,A -90.01312,B 0.00000,C -180.00000} ; preinsert
  LIN {X 9749.966,Y -0.300,Z -43.414,A -90.01312,B 0.00000,C -180.00000} ; insert
  LIN {X 9749.966,Y -0.300,Z -43.414,A -90.01312,B 0.00000,C -180.00000} ; release
  LIN {X 9749.966,Y -0.300,Z 256.586,A -90.01312,B 0.00000,C -180.00000} ; retreat
  ; Step 2767, bar 80
  LIN {X 9874.966,Y -0.300,Z 1164.951,A -90.01312,B 0.00000,C -180.00000} ; outside
  LIN {X 9874.966,Y -0.300,Z 206.586,A -90.01312,B 0.00000,C -180.00000} ; preinsert
  LIN {X 9874.966,Y -0.300,Z -43.414,A -90.01312,B 0.00000,C -180.00000} ; insert
  LIN {X 9874.966,Y -0.300,Z -43.414,A -90.01312,B 0.00000,C -180.00000} ; release
  LIN {X 9874.966,Y -0.300,Z 256.586,A -90.01312,B 0.00000,C -180.00000} ; retreat
  ; Step 2768, bar 81
  LIN {X 10124.966,Y -0.300,Z 1164.951,A -90.01312,B 0.00000,C -180.00000} ; outside
  LIN {X 10124.966,Y -0.300,Z 206.586,A -90.01312,B 0.00000,C -180.00000} ; preinsert
  LIN {X 10124.966,Y -0.300,Z -43.414,A -90.01312,B 0.00000,C -180.00000} ; insert
  LIN {X 10124.966,Y -0.300,Z -43.414,A -90.01312,B 0.00000,C -180.00000} ; release
  LIN {X 10124.966,Y -0.300,Z 256.586,A -90.01312,B 0.00000,C -180.00000} ; retreat
  ; Step 2769, bar 82
  LIN {X 10249.966,Y -0.300,Z 1164.951,A -90.01312,B 0.00000,C -180.00000} ; outside
  LIN {X 10249.966,Y -0.300,Z 206.586,A -90.01312,B 0.00000,C -180.00000} ; preinsert
  LIN {X 10249.966,Y -0.300,Z -43.414,A -90.01312,B 0.00000,C -180.00000} ; insert
  LIN {X 10249.966,Y -0.300,Z -43.414,A -90.01312,B 0.00000,C -180.00000} ; release
  LIN {X 10249.966,Y -0.300,Z 256.586,A -90.01312,B 0.00000,C -180.00000} ; retreat
  ; Step 2770, bar 83
  LIN {X 10374.966,Y -0.300,Z 1164.951,A -90.01312,B 0.00000,C -180.00000} ; outside
  LIN {X 10374.966,Y -0.300,Z 206.586,A -90.01312,B 0.00000,C -180.00000} ; preinsert
  LIN {X 10374.966,Y -0.300,Z -43.414,A -90.01312,B 0.00000,C -180.00000} ; insert
  LIN {X 10374.966,Y -0.300,Z -43.414,A -90.01312,B 0.00000,C -180.00000} ; release
  LIN {X 10374.966,Y -0.300,Z 256.586,A -90.01312,B 0.00000,C -180.00000} ; retreat
  ; Step 2771, bar 84
  LIN {X 10499.966,Y -0.300,Z 1164.951,A -90.01312,B 0.00000,C -180.00000} ; outside
  LIN {X 10499.966,Y -0.300,Z 206.586,A -90.01312,B 0.00000,C -180.00000} ; preinsert
  LIN {X 10499.966,Y -0.300,Z -43.414,A -90.01312,B 0.00000,C -180.00000} ; insert
  LIN {X 10499.966,Y -0.300,Z -43.414,A -90.01312,B 0.00000,C -180.00000} ; release
  LIN {X 10499.966,Y -0.300,Z 256.586,A -90.01312,B 0.00000,C -180.00000} ; retreat
  ; Step 2772, bar 85
  LIN {X 10624.966,Y -0.300,Z 1164.951,A -90.01312,B 0.00000,C -180.00000} ; outside
  LIN {X 10624.966,Y -0.300,Z 206.586,A -90.01312,B 0.00000,C -180.00000} ; preinsert
  LIN {X 10624.966,Y -0.300,Z -43.414,A -90.01312,B 0.00000,C -180.00000} ; insert
  LIN {X 10624.966,Y -0.300,Z -43.414,A -90.01312,B 0.00000,C -180.00000} ; release
  LIN {X 10624.966,Y -0.300,Z 256.586,A -90.01312,B 0.00000,C -180.00000} ; retreat
  ; Step 2773, bar 86
  LIN {X 10749.966,Y -0.300,Z 1164.951,A -90.01312,B 0.00000,C -180.00000} ; outside
  LIN {X 10749.966,Y -0.300,Z 206.586,A -90.01312,B 0.00000,C -180.00000} ; preinsert
  LIN {X 10749.966,Y -0.300,Z -43.414,A -90.01312,B 0.00000,C -180.00000} ; insert
  LIN {X 10749.966,Y -0.300,Z -43.414,A -90.01312,B 0.00000,C -180.00000} ; release
  LIN {X 10749.966,Y -0.300,Z 256.586,A -90.01312,B 0.00000,C -180.00000} ; retreat
  ; Step 2774, bar 87
  LIN {X 10874.966,Y -0.300,Z 1164.951,A -90.01312,B 0.00000,C -180.00000} ; outside
  LIN {X 10874.966,Y -0.300,Z 206.586,A -90.01312,B 0.00000,C -180.00000} ; preinsert
  LIN {X 10874.966,Y -0.300,Z -43.414,A -90.01312,B 0.00000,C -180.00000} ; insert
  LIN {X 10874.966,Y -0.300,Z -43.414,A -90.01312,B 0.00000,C -180.00000} ; release
  LIN {X 10874.966,Y -0.300,Z 256.586,A -90.01312,B 0.00000,C -180.00000} ; retreat
  ; Step 2775, bar 88
  LIN {X 10999.966,Y -0.300,Z 1164.951,A -90.01312,B 0.00000,C -180.00000} ; outside
  LIN {X 10999.966,Y -0.300,Z 206.586,A -90.01312,B 0.00000,C -180.00000} ; preinsert
  LIN {X 10999.966,Y -0.300,Z -43.414,A -90.01312,B 0.00000,C -180.00000} ; insert
  LIN {X 10999.966,Y -0.300,Z -43.414,A -90.01312,B 0.00000,C -180.00000} ; release
  LIN {X 10999.966,Y -0.300,Z 256.586,A -90.01312,B 0.00000,C -180.00000} ; retreat
  ; Step 2776, bar 89
  LIN {X 11124.966,Y -0.300,Z 1164.951,A -90.01312,B 0.00000,C -180.00000} ; outside
  LIN {X 11124.966,Y -0.300,Z 206.586,A -90.01312,B 0.00000,C -180.00000} ; preinsert
  LIN {X 11124.966,Y -0.300,Z -43.414,A -90.01312,B 0.00000,C -180.00000} ; insert
  LIN {X 11124.966,Y -0.300,Z -43.414,A -90.01312,B 0.00000,C -180.00000} ; release
  LIN {X 11124.966,Y -0.300,Z 256.586,A -90.01312,B 0.00000,C -180.00000} ; retreat
  ; Step 2777, bar 90
  LIN {X 11249.966,Y -0.300,Z 1164.951,A -90.01312,B 0.00000,C -180.00000} ; outside
  LIN {X 11249.966,Y -0.300,Z 206.586,A -90.01312,B 0.00000,C -180.00000} ; preinsert
  LIN {X 11249.966,Y -0.300,Z -43.414,A -90.01312,B 0.00000,C -180.00000} ; insert
  LIN {X 11249.966,Y -0.300,Z -43.414,A -90.01312,B 0.00000,C -180.00000} ; release
  LIN {X 11249.966,Y -0.300,Z 256.586,A -90.01312,B 0.00000,C -180.00000} ; retreat
  ; Step 2778, bar 91
  LIN {X 11374.966,Y -0.300,Z 1164.951,A -90.01312,B 0.00000,C -180.00000} ; outside
  LIN {X 11374.966,Y -0.300,Z 206.586,A -90.01312,B 0.00000,C -180.00000} ; preinsert
  LIN {X 11374.966,Y -0.300,Z -43.414,A -90.01312,B 0.00000,C -180.00000} ; insert
  LIN {X 11374.966,Y -0.300,Z -43.414,A -90.01312,B 0.00000,C -180.00000} ; release
  LIN {X 11374.966,Y -0.300,Z 256.586,A -90.01312,B 0.00000,C -180.00000} ; retreat
  ; Step 2779, bar 92
  LIN {X 11499.966,Y -0.300,Z 1164.951,A -90.01312,B 0.00000,C -180.00000} ; outside
  LIN {X 11499.966,Y -0.300,Z 206.586,A -90.01312,B 0.00000,C -180.00000} ; preinsert
  LIN {X 11499.966,Y -0.300,Z -43.414,A -90.01312,B 0.00000,C -180.00000} ; insert
  LIN {X 11499.966,Y -0.300,Z -43.414,A -90.01312,B 0.00000,C -180.00000} ; release
  LIN {X 11499.966,Y -0.300,Z 256.586,A -90.01312,B 0.00000,C -180.00000} ; retreat
  ; Step 2780, bar 93
  LIN {X 11624.966,Y -0.300,Z 1164.951,A -90.01312,B 0.00000,C -180.00000} ; outside
  LIN {X 11624.966,Y -0.300,Z 206.586,A -90.01312,B 0.00000,C -180.00000} ; preinsert
  LIN {X 11624.966,Y -0.300,Z -43.414,A -90.01312,B 0.00000,C -180.00000} ; insert
  LIN {X 11624.966,Y -0.300,Z -43.414,A -90.01312,B 0.00000,C -180.00000} ; release
  LIN {X 11624.966,Y -0.300,Z 256.586,A -90.01312,B 0.00000,C -180.00000} ; retreat
  ; Step 2781, bar 94
  LIN {X 11749.966,Y -0.300,Z 1164.951,A -90.01312,B 0.00000,C -180.00000} ; outside
  LIN {X 11749.966,Y -0.300,Z 206.586,A -90.01312,B 0.00000,C -180.00000} ; preinsert
  LIN {X 11749.966,Y -0.300,Z -43.414,A -90.01312,B 0.00000,C -180.00000} ; insert
  LIN {X 11749.966,Y -0.300,Z -43.414,A -90.01312,B 0.00000,C -180.00000} ; release
  LIN {X 11749.966,Y -0.300,Z 256.586,A -90.01312,B 0.00000,C -180.00000} ; retreat
  ; Step 2782, bar 95
  LIN {X 11874.966,Y -0.300,Z 1164.951,A -90.01312,B 0.00000,C -180.00000} ; outside
  LIN {X 11874.966,Y -0.300,Z 206.586,A -90.01312,B 0.00000,C -180.00000} ; preinsert
  LIN {X 11874.966,Y -0.300,Z -43.414,A -90.01312,B 0.00000,C -180.00000} ; insert
  LIN {X 11874.966,Y -0.300,Z -43.414,A -90.01312,B 0.00000,C -180.00000} ; release
  LIN {X 11874.966,Y -0.300,Z 256.586,A -90.01312,B 0.00000,C -180.00000} ; retreat
  ; Step 2783, bar 96
  LIN {X 11999.966,Y -0.300,Z 1164.951,A -90.01312,B 0.00000,C -180.00000} ; outside
  LIN {X 11999.966,Y -0.300,Z 206.586,A -90.01312,B 0.00000,C -180.00000} ; preinsert
  LIN {X 11999.966,Y -0.300,Z -43.414,A -90.01312,B 0.00000,C -180.00000} ; insert
  LIN {X 11999.966,Y -0.300,Z -43.414,A -90.01312,B 0.00000,C -180.00000} ; release
  LIN {X 11999.966,Y -0.300,Z 256.586,A -90.01312,B 0.00000,C -180.00000} ; retreat
  ; Step 2784, bar 97
  LIN {X 12124.966,Y -0.300,Z 1164.951,A -90.01312,B 0.00000,C -180.00000} ; outside
  LIN {X 12124.966,Y -0.300,Z 206.586,A -90.01312,B 0.00000,C -180.00000} ; preinsert
  LIN {X 12124.966,Y -0.300,Z -43.414,A -90.01312,B 0.00000,C -180.00000} ; insert
  LIN {X 12124.966,Y -0.300,Z -43.414,A -90.01312,B 0.00000,C -180.00000} ; release
  LIN {X 12124.966,Y -0.300,Z 256.586,A -90.01312,B 0.00000,C -180.00000} ; retreat
  ; Step 2785, bar 98
  LIN {X 12249.966,Y -0.300,Z 1164.951,A -90.01312,B 0.00000,C -180.00000} ; outside
  LIN {X 12249.966,Y -0.300,Z 206.586,A -90.01312,B 0.00000,C -180.00000} ; preinsert
  LIN {X 12249.966,Y -0.300,Z -43.414,A -90.01312,B 0.00000,C -180.00000} ; insert
  LIN {X 12249.966,Y -0.300,Z -43.414,A -90.01312,B 0.00000,C -180.00000} ; release
  LIN {X 12249.966,Y -0.300,Z 256.586,A -90.01312,B 0.00000,C -180.00000} ; retreat
  ; Step 2786, bar 99
  LIN {X 12349.966,Y -0.300,Z 1164.951,A -90.01312,B 0.00000,C -180.00000} ; outside
  LIN {X 12349.966,Y -0.300,Z 206.586,A -90.01312,B 0.00000,C -180.00000} ; preinsert
  LIN {X 12349.966,Y -0.300,Z -43.414,A -90.01312,B 0.00000,C -180.00000} ; insert
  LIN {X 12349.966,Y -0.300,Z -43.414,A -90.01312,B 0.00000,C -180.00000} ; release
  LIN {X 12349.966,Y -0.300,Z 256.586,A -90.01312,B 0.00000,C -180.00000} ; retreat
  ; Step 2787, bar 100
  LIN {X 12449.966,Y -0.300,Z 1164.951,A -90.01312,B 0.00000,C -180.00000} ; outside
  LIN {X 12449.966,Y -0.300,Z 206.586,A -90.01312,B 0.00000,C -180.00000} ; preinsert
  LIN {X 12449.966,Y -0.300,Z -43.414,A -90.01312,B 0.00000,C -180.00000} ; insert
  LIN {X 12449.966,Y -0.300,Z -43.414,A -90.01312,B 0.00000,C -180.00000} ; release
  LIN {X 12449.966,Y -0.300,Z 256.586,A -90.01312,B 0.00000,C -180.00000} ; retreat
  ; Step 2788, bar 101
  LIN {X 12549.966,Y -0.300,Z 1164.951,A -90.01312,B 0.00000,C -180.00000} ; outside
  LIN {X 12549.966,Y -0.300,Z 206.586,A -90.01312,B 0.00000,C -180.00000} ; preinsert
  LIN {X 12549.966,Y -0.300,Z -43.414,A -90.01312,B 0.00000,C -180.00000} ; insert
  LIN {X 12549.966,Y -0.300,Z -43.414,A -90.01312,B 0.00000,C -180.00000} ; release
  LIN {X 12549.966,Y -0.300,Z 256.586,A -90.01312,B 0.00000,C -180.00000} ; retreat
  ; Step 2789, bar 102
  LIN {X 12649.966,Y -0.300,Z 1164.951,A -90.01312,B 0.00000,C -180.00000} ; outside
  LIN {X 12649.966,Y -0.300,Z 206.586,A -90.01312,B 0.00000,C -180.00000} ; preinsert
  LIN {X 12649.966,Y -0.300,Z -43.414,A -90.01312,B 0.00000,C -180.00000} ; insert
  LIN {X 12649.966,Y -0.300,Z -43.414,A -90.01312,B 0.00000,C -180.00000} ; release
  LIN {X 12649.966,Y -0.300,Z 256.586,A -90.01312,B 0.00000,C -180.00000} ; retreat
  ; Step 2790, bar 103
  LIN {X 12749.966,Y -0.300,Z 1164.951,A -90.01312,B 0.00000,C -180.00000} ; outside
  LIN {X 12749.966,Y -0.300,Z 206.586,A -90.01312,B 0.00000,C -180.00000} ; preinsert
  LIN {X 12749.966,Y -0.300,Z -43.414,A -90.01312,B 0.00000,C -180.00000} ; insert
  LIN {X 12749.966,Y -0.300,Z -43.414,A -90.01312,B 0.00000,C -180.00000} ; release
  LIN {X 12749.966,Y -0.300,Z 256.586,A -90.01312,B 0.00000,C -180.00000} ; retreat
  ; Step 2791, bar 104
  LIN {X 12849.966,Y -0.300,Z 1164.951,A -90.01312,B 0.00000,C -180.00000} ; outside
  LIN {X 12849.966,Y -0.300,Z 206.586,A -90.01312,B 0.00000,C -180.00000} ; preinsert
  LIN {X 12849.966,Y -0.300,Z -43.414,A -90.01312,B 0.00000,C -180.00000} ; insert
  LIN {X 12849.966,Y -0.300,Z -43.414,A -90.01312,B 0.00000,C -180.00000} ; release
  LIN {X 12849.966,Y -0.300,Z 256.586,A -90.01312,B 0.00000,C -180.00000} ; retreat
  ; Step 2792, bar 105
  LIN {X 12949.966,Y -0.300,Z 1164.951,A -90.01312,B 0.00000,C -180.00000} ; outside
  LIN {X 12949.966,Y -0.300,Z 206.586,A -90.01312,B 0.00000,C -180.00000} ; preinsert
  LIN {X 12949.966,Y -0.300,Z -43.414,A -90.01312,B 0.00000,C -180.00000} ; insert
  LIN {X 12949.966,Y -0.300,Z -43.414,A -90.01312,B 0.00000,C -180.00000} ; release
  LIN {X 12949.966,Y -0.300,Z 256.586,A -90.01312,B 0.00000,C -180.00000} ; retreat
  ; Step 2793, bar 106
  LIN {X 13049.966,Y -0.300,Z 1164.951,A -90.01312,B 0.00000,C -180.00000} ; outside
  LIN {X 13049.966,Y -0.300,Z 206.586,A -90.01312,B 0.00000,C -180.00000} ; preinsert
  LIN {X 13049.966,Y -0.300,Z -43.414,A -90.01312,B 0.00000,C -180.00000} ; insert
  LIN {X 13049.966,Y -0.300,Z -43.414,A -90.01312,B 0.00000,C -180.00000} ; release
  LIN {X 13049.966,Y -0.300,Z 256.586,A -90.01312,B 0.00000,C -180.00000} ; retreat
  ; Step 2794, bar 107
  LIN {X 13149.966,Y -0.300,Z 1164.951,A -90.01312,B 0.00000,C -180.00000} ; outside
  LIN {X 13149.966,Y -0.300,Z 206.586,A -90.01312,B 0.00000,C -180.00000} ; preinsert
  LIN {X 13149.966,Y -0.300,Z -43.414,A -90.01312,B 0.00000,C -180.00000} ; insert
  LIN {X 13149.966,Y -0.300,Z -43.414,A -90.01312,B 0.00000,C -180.00000} ; release
  LIN {X 13149.966,Y -0.300,Z 256.586,A -90.01312,B 0.00000,C -180.00000} ; retreat
  ; Step 2795, bar 108
  LIN {X 13249.966,Y -0.300,Z 1164.951,A -90.01312,B 0.00000,C -180.00000} ; outside
  LIN {X 13249.966,Y -0.300,Z 206.586,A -90.01312,B 0.00000,C -180.00000} ; preinsert
  LIN {X 13249.966,Y -0.300,Z -43.414,A -90.01312,B 0.00000,C -180.00000} ; insert
  LIN {X 13249.966,Y -0.300,Z -43.414,A -90.01312,B 0.00000,C -180.00000} ; release
  LIN {X 13249.966,Y -0.300,Z 256.586,A -90.01312,B 0.00000,C -180.00000} ; retreat
  ; Step 2796, bar 109
  LIN {X 13349.966,Y -0.300,Z 1164.951,A -90.01312,B 0.00000,C -180.00000} ; outside
  LIN {X 13349.966,Y -0.300,Z 206.586,A -90.01312,B 0.00000,C -180.00000} ; preinsert
  LIN {X 13349.966,Y -0.300,Z -43.414,A -90.01312,B 0.00000,C -180.00000} ; insert
  LIN {X 13349.966,Y -0.300,Z -43.414,A -90.01312,B 0.00000,C -180.00000} ; release
  LIN {X 13349.966,Y -0.300,Z 256.586,A -90.01312,B 0.00000,C -180.00000} ; retreat
  ; Step 2797, bar 110
  LIN {X 13449.966,Y -0.300,Z 1164.951,A -90.01312,B 0.00000,C -180.00000} ; outside
  LIN {X 13449.966,Y -0.300,Z 206.586,A -90.01312,B 0.00000,C -180.00000} ; preinsert
  LIN {X 13449.966,Y -0.300,Z -43.414,A -90.01312,B 0.00000,C -180.00000} ; insert
  LIN {X 13449.966,Y -0.300,Z -43.414,A -90.01312,B 0.00000,C -180.00000} ; release
  LIN {X 13449.966,Y -0.300,Z 256.586,A -90.01312,B 0.00000,C -180.00000} ; retreat
  ; Step 2798, bar 111
  LIN {X 13549.966,Y -0.300,Z 1164.951,A -90.01312,B 0.00000,C -180.00000} ; outside
  LIN {X 13549.966,Y -0.300,Z 206.586,A -90.01312,B 0.00000,C -180.00000} ; preinsert
  LIN {X 13549.966,Y -0.300,Z -43.414,A -90.01312,B 0.00000,C -180.00000} ; insert
  LIN {X 13549.966,Y -0.300,Z -43.414,A -90.01312,B 0.00000,C -180.00000} ; release
  LIN {X 13549.966,Y -0.300,Z 256.586,A -90.01312,B 0.00000,C -180.00000} ; retreat
  ; Step 2799, bar 112
  LIN {X 13649.966,Y -0.300,Z 1164.951,A -90.01312,B 0.00000,C -180.00000} ; outside
  LIN {X 13649.966,Y -0.300,Z 206.586,A -90.01312,B 0.00000,C -180.00000} ; preinsert
  LIN {X 13649.966,Y -0.300,Z -43.414,A -90.01312,B 0.00000,C -180.00000} ; insert
  LIN {X 13649.966,Y -0.300,Z -43.414,A -90.01312,B 0.00000,C -180.00000} ; release
  LIN {X 13649.966,Y -0.300,Z 256.586,A -90.01312,B 0.00000,C -180.00000} ; retreat
  ; Step 2800, bar 274
  LIN {X -14049.896,Y 0.264,Z 1163.390,A -90.00000,B 0.00000,C -180.00000} ; outside
  LIN {X -14049.896,Y 0.264,Z 205.570,A -90.00000,B 0.00000,C -180.00000} ; preinsert
  LIN {X -14049.896,Y 0.264,Z -44.430,A -90.00000,B 0.00000,C -180.00000} ; insert
  LIN {X -14049.896,Y 0.264,Z -44.430,A -90.00000,B 0.00000,C -180.00000} ; release
  LIN {X -14049.896,Y 0.264,Z 255.570,A -90.00000,B 0.00000,C -180.00000} ; retreat
  ; Step 2801, bar 273
  LIN {X -13949.896,Y 0.264,Z 1163.390,A -90.00000,B 0.00000,C -180.00000} ; outside
  LIN {X -13949.896,Y 0.264,Z 205.570,A -90.00000,B 0.00000,C -180.00000} ; preinsert
  LIN {X -13949.896,Y 0.264,Z -44.430,A -90.00000,B 0.00000,C -180.00000} ; insert
  LIN {X -13949.896,Y 0.264,Z -44.430,A -90.00000,B 0.00000,C -180.00000} ; release
  LIN {X -13949.896,Y 0.264,Z 255.570,A -90.00000,B 0.00000,C -180.00000} ; retreat
  ; Step 2802, bar 115
  LIN {X 13949.896,Y 0.264,Z 1163.390,A -90.00000,B 0.00000,C 180.00000} ; outside
  LIN {X 13949.896,Y 0.264,Z 205.570,A -90.00000,B 0.00000,C 180.00000} ; preinsert
  LIN {X 13949.896,Y 0.264,Z -44.430,A -90.00000,B 0.00000,C 180.00000} ; insert
  LIN {X 13949.896,Y 0.264,Z -44.430,A -90.00000,B 0.00000,C 180.00000} ; release
  LIN {X 13949.896,Y 0.264,Z 255.570,A -90.00000,B 0.00000,C 180.00000} ; retreat
  ; Step 2803, bar 116
  LIN {X 14049.896,Y 0.264,Z 1163.390,A -90.00000,B 0.00000,C 180.00000} ; outside
  LIN {X 14049.896,Y 0.264,Z 205.570,A -90.00000,B 0.00000,C 180.00000} ; preinsert
  LIN {X 14049.896,Y 0.264,Z -44.430,A -90.00000,B 0.00000,C 180.00000} ; insert
  LIN {X 14049.896,Y 0.264,Z -44.430,A -90.00000,B 0.00000,C 180.00000} ; release
  LIN {X 14049.896,Y 0.264,Z 255.570,A -90.00000,B 0.00000,C 180.00000} ; retreat
  ; Step 2804, bar 121
  LIN {X 14550.194,Y -0.251,Z 1164.434,A -90.04135,B 0.00000,C -180.00000} ; outside
  LIN {X 14550.194,Y -0.251,Z 206.506,A -90.04135,B 0.00000,C -180.00000} ; preinsert
  LIN {X 14550.194,Y -0.251,Z -43.494,A -90.04135,B 0.00000,C -180.00000} ; insert
  LIN {X 14550.194,Y -0.251,Z -43.494,A -90.04135,B 0.00000,C -180.00000} ; release
  LIN {X 14550.194,Y -0.251,Z 256.506,A -90.04135,B 0.00000,C -180.00000} ; retreat
  ; Step 2805, bar 131
  LIN {X 15550.194,Y -0.251,Z 1164.434,A -90.04135,B 0.00000,C -180.00000} ; outside
  LIN {X 15550.194,Y -0.251,Z 206.506,A -90.04135,B 0.00000,C -180.00000} ; preinsert
  LIN {X 15550.194,Y -0.251,Z -43.494,A -90.04135,B 0.00000,C -180.00000} ; insert
  LIN {X 15550.194,Y -0.251,Z -43.494,A -90.04135,B 0.00000,C -180.00000} ; release
  LIN {X 15550.194,Y -0.251,Z 256.506,A -90.04135,B 0.00000,C -180.00000} ; retreat
  ; Step 2806, bar 1858
  LIN {X -15549.931,Y 0.371,Z 795.552,A 89.99798,B 0.00000,C -180.00000} ; outside
  LIN {X -15549.931,Y 0.371,Z -167.271,A 89.99798,B 0.00000,C -180.00000} ; preinsert
  LIN {X -15549.931,Y 0.371,Z -417.271,A 89.99798,B 0.00000,C -180.00000} ; insert
  LIN {X -15549.931,Y 0.371,Z -417.271,A 89.99798,B 0.00000,C -180.00000} ; release
  LIN {X -15549.931,Y 0.371,Z -117.271,A 89.99798,B 0.00000,C -180.00000} ; retreat
  ; Step 2807, bar 1054
  LIN {X 15549.931,Y 0.371,Z 795.552,A 90.00202,B 0.00000,C 180.00000} ; outside
  LIN {X 15549.931,Y 0.371,Z -167.271,A 90.00202,B 0.00000,C 180.00000} ; preinsert
  LIN {X 15549.931,Y 0.371,Z -417.271,A 90.00202,B 0.00000,C 180.00000} ; insert
  LIN {X 15549.931,Y 0.371,Z -417.271,A 90.00202,B 0.00000,C 180.00000} ; release
  LIN {X 15549.931,Y 0.371,Z -117.271,A 90.00202,B 0.00000,C 180.00000} ; retreat
  ; Step 2808, bar 3017
  LIN {X 14849.996,Y -231.529,Z 999.147,A -7.53655,B 0.00000,C 180.00000} ; outside
  LIN {X 14849.996,Y -231.529,Z 33.662,A -7.53655,B 0.00000,C 180.00000} ; preinsert
  LIN {X 14849.996,Y -231.529,Z -216.338,A -7.53655,B 0.00000,C 180.00000} ; insert
  LIN {X 14849.996,Y -231.529,Z -216.338,A -7.53655,B 0.00000,C 180.00000} ; release
  LIN {X 14849.996,Y -231.529,Z 83.662,A -7.53655,B 0.00000,C 180.00000} ; retreat
  ; Step 2809, bar 2978
  LIN {X -14849.996,Y -231.529,Z 999.139,A -172.46345,B 0.00000,C -180.00000} ; outside
  LIN {X -14849.996,Y -231.529,Z 33.655,A -172.46345,B 0.00000,C -180.00000} ; preinsert
  LIN {X -14849.996,Y -231.529,Z -216.345,A -172.46345,B 0.00000,C -180.00000} ; insert
  LIN {X -14849.996,Y -231.529,Z -216.345,A -172.46345,B 0.00000,C -180.00000} ; release
  LIN {X -14849.996,Y -231.529,Z 83.655,A -172.46345,B 0.00000,C -180.00000} ; retreat
  ; Step 2810, bar 2960
  LIN {X -14849.996,Y 231.529,Z 999.147,A 172.46345,B 0.00000,C 180.00000} ; outside
  LIN {X -14849.996,Y 231.529,Z 33.662,A 172.46345,B 0.00000,C 180.00000} ; preinsert
  LIN {X -14849.996,Y 231.529,Z -216.338,A 172.46345,B 0.00000,C 180.00000} ; insert
  LIN {X -14849.996,Y 231.529,Z -216.338,A 172.46345,B 0.00000,C 180.00000} ; release
  LIN {X -14849.996,Y 231.529,Z 83.662,A 172.46345,B 0.00000,C 180.00000} ; retreat
  ; Step 2811, bar 2999
  LIN {X 14849.996,Y 231.529,Z 999.139,A 7.53655,B 0.00000,C 180.00000} ; outside
  LIN {X 14849.996,Y 231.529,Z 33.655,A 7.53655,B 0.00000,C 180.00000} ; preinsert
  LIN {X 14849.996,Y 231.529,Z -216.345,A 7.53655,B 0.00000,C 180.00000} ; insert
  LIN {X 14849.996,Y 231.529,Z -216.345,A 7.53655,B 0.00000,C 180.00000} ; release
  LIN {X 14849.996,Y 231.529,Z 83.655,A 7.53655,B 0.00000,C 180.00000} ; retreat
  ; Step 2812, bar 2996
  LIN {X 14450.033,Y -18.400,Z 1015.810,A -48.70858,B 0.00000,C 180.00000} ; outside
  LIN {X 14450.033,Y -18.400,Z 49.700,A -48.70858,B 0.00000,C 180.00000} ; preinsert
  LIN {X 14450.033,Y -18.400,Z -200.300,A -48.70858,B 0.00000,C 180.00000} ; insert
  LIN {X 14450.033,Y -18.400,Z -200.300,A -48.70858,B 0.00000,C 180.00000} ; release
  LIN {X 14450.033,Y -18.400,Z 99.700,A -48.70858,B 0.00000,C 180.00000} ; retreat
  ; Step 2813, bar 2957
  LIN {X -14450.033,Y -18.400,Z 1015.810,A -131.29142,B 0.00000,C -180.00000} ; outside
  LIN {X -14450.033,Y -18.400,Z 49.700,A -131.29142,B 0.00000,C -180.00000} ; preinsert
  LIN {X -14450.033,Y -18.400,Z -200.300,A -131.29142,B 0.00000,C -180.00000} ; insert
  LIN {X -14450.033,Y -18.400,Z -200.300,A -131.29142,B 0.00000,C -180.00000} ; release
  LIN {X -14450.033,Y -18.400,Z 99.700,A -131.29142,B 0.00000,C -180.00000} ; retreat
  ; Step 2814, bar 3012
  LIN {X 14050.033,Y -231.600,Z 1018.153,A 48.70858,B 0.00000,C 180.00000} ; outside
  LIN {X 14050.033,Y -231.600,Z 52.668,A 48.70858,B 0.00000,C 180.00000} ; preinsert
  LIN {X 14050.033,Y -231.600,Z -197.332,A 48.70858,B 0.00000,C 180.00000} ; insert
  LIN {X 14050.033,Y -231.600,Z -197.332,A 48.70858,B 0.00000,C 180.00000} ; release
  LIN {X 14050.033,Y -231.600,Z 102.668,A 48.70858,B 0.00000,C 180.00000} ; retreat
  ; Step 2815, bar 2954
  LIN {X -14050.033,Y 231.600,Z 1018.153,A -131.29142,B 0.00000,C -180.00000} ; outside
  LIN {X -14050.033,Y 231.600,Z 52.668,A -131.29142,B 0.00000,C -180.00000} ; preinsert
  LIN {X -14050.033,Y 231.600,Z -197.332,A -131.29142,B 0.00000,C -180.00000} ; insert
  LIN {X -14050.033,Y 231.600,Z -197.332,A -131.29142,B 0.00000,C -180.00000} ; release
  LIN {X -14050.033,Y 231.600,Z 102.668,A -131.29142,B 0.00000,C -180.00000} ; retreat
  ; Step 2816, bar 2973
  LIN {X -14050.033,Y -231.600,Z 1018.153,A 131.29142,B 0.00000,C 180.00000} ; outside
  LIN {X -14050.033,Y -231.600,Z 52.668,A 131.29142,B 0.00000,C 180.00000} ; preinsert
  LIN {X -14050.033,Y -231.600,Z -197.332,A 131.29142,B 0.00000,C 180.00000} ; insert
  LIN {X -14050.033,Y -231.600,Z -197.332,A 131.29142,B 0.00000,C 180.00000} ; release
  LIN {X -14050.033,Y -231.600,Z 102.668,A 131.29142,B 0.00000,C 180.00000} ; retreat
  ; Step 2817, bar 2993
  LIN {X 14050.033,Y 231.600,Z 1018.153,A -48.70858,B 0.00000,C 180.00000} ; outside
  LIN {X 14050.033,Y 231.600,Z 52.668,A -48.70858,B 0.00000,C 180.00000} ; preinsert
  LIN {X 14050.033,Y 231.600,Z -197.332,A -48.70858,B 0.00000,C 180.00000} ; insert
  LIN {X 14050.033,Y 231.600,Z -197.332,A -48.70858,B 0.00000,C 180.00000} ; release
  LIN {X 14050.033,Y 231.600,Z 102.668,A -48.70858,B 0.00000,C 180.00000} ; retreat
  ; Step 2818, bar 2951
  LIN {X -13650.008,Y -18.390,Z 1034.171,A -90.84847,B 0.00000,C -180.00000} ; outside
  LIN {X -13650.008,Y -18.390,Z 68.062,A -90.84847,B 0.00000,C -180.00000} ; preinsert
  LIN {X -13650.008,Y -18.390,Z -181.938,A -90.84847,B 0.00000,C -180.00000} ; insert
  LIN {X -13650.008,Y -18.390,Z -181.938,A -90.84847,B 0.00000,C -180.00000} ; release
  LIN {X -13650.008,Y -18.390,Z 118.062,A -90.84847,B 0.00000,C -180.00000} ; retreat
  ; Step 2819, bar 2990
  LIN {X 13650.008,Y -18.390,Z 1034.171,A -89.15153,B 0.00000,C -180.00000} ; outside
  LIN {X 13650.008,Y -18.390,Z 68.062,A -89.15153,B 0.00000,C -180.00000} ; preinsert
  LIN {X 13650.008,Y -18.390,Z -181.938,A -89.15153,B 0.00000,C -180.00000} ; insert
  LIN {X 13650.008,Y -18.390,Z -181.938,A -89.15153,B 0.00000,C -180.00000} ; release
  LIN {X 13650.008,Y -18.390,Z 118.062,A -89.15153,B 0.00000,C -180.00000} ; retreat
  ; Step 2820, bar 3007
  LIN {X 13249.942,Y -231.601,Z 1051.450,A 88.44949,B 0.00000,C 180.00000} ; outside
  LIN {X 13249.942,Y -231.601,Z 85.965,A 88.44949,B 0.00000,C 180.00000} ; preinsert
  LIN {X 13249.942,Y -231.601,Z -164.035,A 88.44949,B 0.00000,C 180.00000} ; insert
  LIN {X 13249.942,Y -231.601,Z -164.035,A 88.44949,B 0.00000,C 180.00000} ; release
  LIN {X 13249.942,Y -231.601,Z 135.965,A 88.44949,B 0.00000,C 180.00000} ; retreat
  ; Step 2821, bar 2968
  LIN {X -13249.942,Y -231.601,Z 1051.450,A 91.55051,B 0.00000,C 180.00000} ; outside
  LIN {X -13249.942,Y -231.601,Z 85.965,A 91.55051,B 0.00000,C 180.00000} ; preinsert
  LIN {X -13249.942,Y -231.601,Z -164.035,A 91.55051,B 0.00000,C 180.00000} ; insert
  LIN {X -13249.942,Y -231.601,Z -164.035,A 91.55051,B 0.00000,C 180.00000} ; release
  LIN {X -13249.942,Y -231.601,Z 135.965,A 91.55051,B 0.00000,C 180.00000} ; retreat
  ; Step 2822, bar 2948
  LIN {X -13249.942,Y 231.601,Z 1051.450,A -91.55051,B 0.00000,C -180.00000} ; outside
  LIN {X -13249.942,Y 231.601,Z 85.965,A -91.55051,B 0.00000,C -180.00000} ; preinsert
  LIN {X -13249.942,Y 231.601,Z -164.035,A -91.55051,B 0.00000,C -180.00000} ; insert
  LIN {X -13249.942,Y 231.601,Z -164.035,A -91.55051,B 0.00000,C -180.00000} ; release
  LIN {X -13249.942,Y 231.601,Z 135.965,A -91.55051,B 0.00000,C -180.00000} ; retreat
  ; Step 2823, bar 2987
  LIN {X 13249.942,Y 231.601,Z 1051.450,A -88.44949,B 0.00000,C 180.00000} ; outside
  LIN {X 13249.942,Y 231.601,Z 85.965,A -88.44949,B 0.00000,C 180.00000} ; preinsert
  LIN {X 13249.942,Y 231.601,Z -164.035,A -88.44949,B 0.00000,C 180.00000} ; insert
  LIN {X 13249.942,Y 231.601,Z -164.035,A -88.44949,B 0.00000,C 180.00000} ; release
  LIN {X 13249.942,Y 231.601,Z 135.965,A -88.44949,B 0.00000,C 180.00000} ; retreat
  ; Step 2824, bar 2945
  LIN {X -12850.007,Y -18.193,Z 1068.873,A -90.84369,B 0.00000,C 180.00000} ; outside
  LIN {X -12850.007,Y -18.193,Z 102.763,A -90.84369,B 0.00000,C 180.00000} ; preinsert
  LIN {X -12850.007,Y -18.193,Z -147.237,A -90.84369,B 0.00000,C 180.00000} ; insert
  LIN {X -12850.007,Y -18.193,Z -147.237,A -90.84369,B 0.00000,C 180.00000} ; release
  LIN {X -12850.007,Y -18.193,Z 152.763,A -90.84369,B 0.00000,C 180.00000} ; retreat
  ; Step 2825, bar 2984
  LIN {X 12850.007,Y -18.193,Z 1068.873,A -89.15631,B 0.00000,C 180.00000} ; outside
  LIN {X 12850.007,Y -18.193,Z 102.763,A -89.15631,B 0.00000,C 180.00000} ; preinsert
  LIN {X 12850.007,Y -18.193,Z -147.237,A -89.15631,B 0.00000,C 180.00000} ; insert
  LIN {X 12850.007,Y -18.193,Z -147.237,A -89.15631,B 0.00000,C 180.00000} ; release
  LIN {X 12850.007,Y -18.193,Z 152.763,A -89.15631,B 0.00000,C 180.00000} ; retreat
  ; Step 2826, bar 3021
  LIN {X 12450.007,Y -731.800,Z 1073.597,A 89.15631,B 0.00000,C 180.00000} ; outside
  LIN {X 12450.007,Y -731.800,Z 108.113,A 89.15631,B 0.00000,C 180.00000} ; preinsert
  LIN {X 12450.007,Y -731.800,Z -141.887,A 89.15631,B 0.00000,C 180.00000} ; insert
  LIN {X 12450.007,Y -731.800,Z -141.887,A 89.15631,B 0.00000,C 180.00000} ; release
  LIN {X 12450.007,Y -731.800,Z 158.113,A 89.15631,B 0.00000,C 180.00000} ; retreat
  ; Step 2827, bar 2982
  LIN {X -12450.007,Y -731.800,Z 1073.597,A 90.84369,B 0.00000,C -180.00000} ; outside
  LIN {X -12450.007,Y -731.800,Z 108.113,A 90.84369,B 0.00000,C -180.00000} ; preinsert
  LIN {X -12450.007,Y -731.800,Z -141.887,A 90.84369,B 0.00000,C -180.00000} ; insert
  LIN {X -12450.007,Y -731.800,Z -141.887,A 90.84369,B 0.00000,C -180.00000} ; release
  LIN {X -12450.007,Y -731.800,Z 158.113,A 90.84369,B 0.00000,C -180.00000} ; retreat
  ; Step 2828, bar 2964
  LIN {X -12450.007,Y 731.800,Z 1073.597,A -90.84369,B 0.00000,C 180.00000} ; outside
  LIN {X -12450.007,Y 731.800,Z 108.113,A -90.84369,B 0.00000,C 180.00000} ; preinsert
  LIN {X -12450.007,Y 731.800,Z -141.887,A -90.84369,B 0.00000,C 180.00000} ; insert
  LIN {X -12450.007,Y 731.800,Z -141.887,A -90.84369,B 0.00000,C 180.00000} ; release
  LIN {X -12450.007,Y 731.800,Z 158.113,A -90.84369,B 0.00000,C 180.00000} ; retreat
  ; Step 2829, bar 3003
  LIN {X 12450.007,Y 731.800,Z 1073.597,A -89.15631,B 0.00000,C 180.00000} ; outside
  LIN {X 12450.007,Y 731.800,Z 108.113,A -89.15631,B 0.00000,C 180.00000} ; preinsert
  LIN {X 12450.007,Y 731.800,Z -141.887,A -89.15631,B 0.00000,C 180.00000} ; insert
  LIN {X 12450.007,Y 731.800,Z -141.887,A -89.15631,B 0.00000,C 180.00000} ; release
  LIN {X 12450.007,Y 731.800,Z 158.113,A -89.15631,B 0.00000,C 180.00000} ; retreat
  ; Step 2830, bar 2981
  LIN {X -12450.007,Y -231.800,Z 1073.597,A 90.84369,B 0.00000,C -180.00000} ; outside
  LIN {X -12450.007,Y -231.800,Z 108.113,A 90.84369,B 0.00000,C -180.00000} ; preinsert
  LIN {X -12450.007,Y -231.800,Z -141.887,A 90.84369,B 0.00000,C -180.00000} ; insert
  LIN {X -12450.007,Y -231.800,Z -141.887,A 90.84369,B 0.00000,C -180.00000} ; release
  LIN {X -12450.007,Y -231.800,Z 158.113,A 90.84369,B 0.00000,C -180.00000} ; retreat
  ; Step 2831, bar 3002
  LIN {X 12450.007,Y 231.800,Z 1073.597,A -89.15631,B 0.00000,C 180.00000} ; outside
  LIN {X 12450.007,Y 231.800,Z 108.113,A -89.15631,B 0.00000,C 180.00000} ; preinsert
  LIN {X 12450.007,Y 231.800,Z -141.887,A -89.15631,B 0.00000,C 180.00000} ; insert
  LIN {X 12450.007,Y 231.800,Z -141.887,A -89.15631,B 0.00000,C 180.00000} ; release
  LIN {X 12450.007,Y 231.800,Z 158.113,A -89.15631,B 0.00000,C 180.00000} ; retreat
  ; Step 2832, bar 3020
  LIN {X 12450.007,Y -231.800,Z 1073.597,A 89.15631,B 0.00000,C 180.00000} ; outside
  LIN {X 12450.007,Y -231.800,Z 108.113,A 89.15631,B 0.00000,C 180.00000} ; preinsert
  LIN {X 12450.007,Y -231.800,Z -141.887,A 89.15631,B 0.00000,C 180.00000} ; insert
  LIN {X 12450.007,Y -231.800,Z -141.887,A 89.15631,B 0.00000,C 180.00000} ; release
  LIN {X 12450.007,Y -231.800,Z 158.113,A 89.15631,B 0.00000,C 180.00000} ; retreat
  ; Step 2833, bar 2963
  LIN {X -12450.007,Y 231.800,Z 1073.597,A -90.84369,B 0.00000,C 180.00000} ; outside
  LIN {X -12450.007,Y 231.800,Z 108.113,A -90.84369,B 0.00000,C 180.00000} ; preinsert
  LIN {X -12450.007,Y 231.800,Z -141.887,A -90.84369,B 0.00000,C 180.00000} ; insert
  LIN {X -12450.007,Y 231.800,Z -141.887,A -90.84369,B 0.00000,C 180.00000} ; release
  LIN {X -12450.007,Y 231.800,Z 158.113,A -90.84369,B 0.00000,C 180.00000} ; retreat
  ; Step 2834, bar 2892
  LIN {X -11624.916,Y -231.794,Z 1086.991,A 87.44234,B 0.00000,C 180.00000} ; outside
  LIN {X -11624.916,Y -231.794,Z 121.006,A 87.44234,B 0.00000,C 180.00000} ; preinsert
  LIN {X -11624.916,Y -231.794,Z -128.994,A 87.44234,B 0.00000,C 180.00000} ; insert
  LIN {X -11624.916,Y -231.794,Z -128.994,A 87.44234,B 0.00000,C 180.00000} ; release
  LIN {X -11624.916,Y -231.794,Z 171.006,A 87.44234,B 0.00000,C 180.00000} ; retreat
  ; Step 2835, bar 2889
  LIN {X -10874.916,Y -231.794,Z 1086.991,A 87.44234,B 0.00000,C 180.00000} ; outside
  LIN {X -10874.916,Y -231.794,Z 121.006,A 87.44234,B 0.00000,C 180.00000} ; preinsert
  LIN {X -10874.916,Y -231.794,Z -128.994,A 87.44234,B 0.00000,C 180.00000} ; insert
  LIN {X -10874.916,Y -231.794,Z -128.994,A 87.44234,B 0.00000,C 180.00000} ; release
  LIN {X -10874.916,Y -231.794,Z 171.006,A 87.44234,B 0.00000,C 180.00000} ; retreat
  ; Step 2836, bar 2886
  LIN {X -10124.916,Y -231.794,Z 1086.991,A 87.44234,B 0.00000,C 180.00000} ; outside
  LIN {X -10124.916,Y -231.794,Z 121.006,A 87.44234,B 0.00000,C 180.00000} ; preinsert
  LIN {X -10124.916,Y -231.794,Z -128.994,A 87.44234,B 0.00000,C 180.00000} ; insert
  LIN {X -10124.916,Y -231.794,Z -128.994,A 87.44234,B 0.00000,C 180.00000} ; release
  LIN {X -10124.916,Y -231.794,Z 171.006,A 87.44234,B 0.00000,C 180.00000} ; retreat
  ; Step 2837, bar 2883
  LIN {X -9374.916,Y -231.794,Z 1086.991,A 87.44234,B 0.00000,C 180.00000} ; outside
  LIN {X -9374.916,Y -231.794,Z 121.006,A 87.44234,B 0.00000,C 180.00000} ; preinsert
  LIN {X -9374.916,Y -231.794,Z -128.994,A 87.44234,B 0.00000,C 180.00000} ; insert
  LIN {X -9374.916,Y -231.794,Z -128.994,A 87.44234,B 0.00000,C 180.00000} ; release
  LIN {X -9374.916,Y -231.794,Z 171.006,A 87.44234,B 0.00000,C 180.00000} ; retreat
  ; Step 2838, bar 2880
  LIN {X -8624.916,Y -231.794,Z 1086.991,A 87.44234,B 0.00000,C 180.00000} ; outside
  LIN {X -8624.916,Y -231.794,Z 121.006,A 87.44234,B 0.00000,C 180.00000} ; preinsert
  LIN {X -8624.916,Y -231.794,Z -128.994,A 87.44234,B 0.00000,C 180.00000} ; insert
  LIN {X -8624.916,Y -231.794,Z -128.994,A 87.44234,B 0.00000,C 180.00000} ; release
  LIN {X -8624.916,Y -231.794,Z 171.006,A 87.44234,B 0.00000,C 180.00000} ; retreat
  ; Step 2839, bar 2877
  LIN {X -7874.916,Y -231.794,Z 1086.991,A 87.44234,B 0.00000,C 180.00000} ; outside
  LIN {X -7874.916,Y -231.794,Z 121.006,A 87.44234,B 0.00000,C 180.00000} ; preinsert
  LIN {X -7874.916,Y -231.794,Z -128.994,A 87.44234,B 0.00000,C 180.00000} ; insert
  LIN {X -7874.916,Y -231.794,Z -128.994,A 87.44234,B 0.00000,C 180.00000} ; release
  LIN {X -7874.916,Y -231.794,Z 171.006,A 87.44234,B 0.00000,C 180.00000} ; retreat
  ; Step 2840, bar 2874
  LIN {X -7124.916,Y -231.794,Z 1086.991,A 87.44234,B 0.00000,C 180.00000} ; outside
  LIN {X -7124.916,Y -231.794,Z 121.006,A 87.44234,B 0.00000,C 180.00000} ; preinsert
  LIN {X -7124.916,Y -231.794,Z -128.994,A 87.44234,B 0.00000,C 180.00000} ; insert
  LIN {X -7124.916,Y -231.794,Z -128.994,A 87.44234,B 0.00000,C 180.00000} ; release
  LIN {X -7124.916,Y -231.794,Z 171.006,A 87.44234,B 0.00000,C 180.00000} ; retreat
  ; Step 2841, bar 2871
  LIN {X -6374.916,Y -231.794,Z 1086.991,A 87.44234,B 0.00000,C 180.00000} ; outside
  LIN {X -6374.916,Y -231.794,Z 121.006,A 87.44234,B 0.00000,C 180.00000} ; preinsert
  LIN {X -6374.916,Y -231.794,Z -128.994,A 87.44234,B 0.00000,C 180.00000} ; insert
  LIN {X -6374.916,Y -231.794,Z -128.994,A 87.44234,B 0.00000,C 180.00000} ; release
  LIN {X -6374.916,Y -231.794,Z 171.006,A 87.44234,B 0.00000,C 180.00000} ; retreat
  ; Step 2842, bar 2868
  LIN {X -5624.916,Y -231.794,Z 1086.991,A 87.44234,B 0.00000,C 180.00000} ; outside
  LIN {X -5624.916,Y -231.794,Z 121.006,A 87.44234,B 0.00000,C 180.00000} ; preinsert
  LIN {X -5624.916,Y -231.794,Z -128.994,A 87.44234,B 0.00000,C 180.00000} ; insert
  LIN {X -5624.916,Y -231.794,Z -128.994,A 87.44234,B 0.00000,C 180.00000} ; release
  LIN {X -5624.916,Y -231.794,Z 171.006,A 87.44234,B 0.00000,C 180.00000} ; retreat
  ; Step 2843, bar 2865
  LIN {X -4874.916,Y -231.794,Z 1086.991,A 87.44234,B 0.00000,C 180.00000} ; outside
  LIN {X -4874.916,Y -231.794,Z 121.006,A 87.44234,B 0.00000,C 180.00000} ; preinsert
  LIN {X -4874.916,Y -231.794,Z -128.994,A 87.44234,B 0.00000,C 180.00000} ; insert
  LIN {X -4874.916,Y -231.794,Z -128.994,A 87.44234,B 0.00000,C 180.00000} ; release
  LIN {X -4874.916,Y -231.794,Z 171.006,A 87.44234,B 0.00000,C 180.00000} ; retreat
  ; Step 2844, bar 2862
  LIN {X -4124.916,Y -231.794,Z 1086.991,A 87.44234,B 0.00000,C 180.00000} ; outside
  LIN {X -4124.916,Y -231.794,Z 121.006,A 87.44234,B 0.00000,C 180.00000} ; preinsert
  LIN {X -4124.916,Y -231.794,Z -128.994,A 87.44234,B 0.00000,C 180.00000} ; insert
  LIN {X -4124.916,Y -231.794,Z -128.994,A 87.44234,B 0.00000,C 180.00000} ; release
  LIN {X -4124.916,Y -231.794,Z 171.006,A 87.44234,B 0.00000,C 180.00000} ; retreat
  ; Step 2845, bar 2859
  LIN {X -3374.916,Y -231.794,Z 1086.991,A 87.44234,B 0.00000,C 180.00000} ; outside
  LIN {X -3374.916,Y -231.794,Z 121.006,A 87.44234,B 0.00000,C 180.00000} ; preinsert
  LIN {X -3374.916,Y -231.794,Z -128.994,A 87.44234,B 0.00000,C 180.00000} ; insert
  LIN {X -3374.916,Y -231.794,Z -128.994,A 87.44234,B 0.00000,C 180.00000} ; release
  LIN {X -3374.916,Y -231.794,Z 171.006,A 87.44234,B 0.00000,C 180.00000} ; retreat
  ; Step 2846, bar 2856
  LIN {X -2624.916,Y -231.794,Z 1086.991,A 87.44234,B 0.00000,C 180.00000} ; outside
  LIN {X -2624.916,Y -231.794,Z 121.006,A 87.44234,B 0.00000,C 180.00000} ; preinsert
  LIN {X -2624.916,Y -231.794,Z -128.994,A 87.44234,B 0.00000,C 180.00000} ; insert
  LIN {X -2624.916,Y -231.794,Z -128.994,A 87.44234,B 0.00000,C 180.00000} ; release
  LIN {X -2624.916,Y -231.794,Z 171.006,A 87.44234,B 0.00000,C 180.00000} ; retreat
  ; Step 2847, bar 2853
  LIN {X -1874.916,Y -231.794,Z 1086.991,A 87.44234,B 0.00000,C 180.00000} ; outside
  LIN {X -1874.916,Y -231.794,Z 121.006,A 87.44234,B 0.00000,C 180.00000} ; preinsert
  LIN {X -1874.916,Y -231.794,Z -128.994,A 87.44234,B 0.00000,C 180.00000} ; insert
  LIN {X -1874.916,Y -231.794,Z -128.994,A 87.44234,B 0.00000,C 180.00000} ; release
  LIN {X -1874.916,Y -231.794,Z 171.006,A 87.44234,B 0.00000,C 180.00000} ; retreat
  ; Step 2848, bar 2850
  LIN {X -1124.916,Y -231.794,Z 1086.991,A 87.44234,B 0.00000,C 180.00000} ; outside
  LIN {X -1124.916,Y -231.794,Z 121.006,A 87.44234,B 0.00000,C 180.00000} ; preinsert
  LIN {X -1124.916,Y -231.794,Z -128.994,A 87.44234,B 0.00000,C 180.00000} ; insert
  LIN {X -1124.916,Y -231.794,Z -128.994,A 87.44234,B 0.00000,C 180.00000} ; release
  LIN {X -1124.916,Y -231.794,Z 171.006,A 87.44234,B 0.00000,C 180.00000} ; retreat
  ; Step 2849, bar 2847
  LIN {X -374.916,Y -231.794,Z 1086.991,A 87.44234,B 0.00000,C 180.00000} ; outside
  LIN {X -374.916,Y -231.794,Z 121.006,A 87.44234,B 0.00000,C 180.00000} ; preinsert
  LIN {X -374.916,Y -231.794,Z -128.994,A 87.44234,B 0.00000,C 180.00000} ; insert
  LIN {X -374.916,Y -231.794,Z -128.994,A 87.44234,B 0.00000,C 180.00000} ; release
  LIN {X -374.916,Y -231.794,Z 171.006,A 87.44234,B 0.00000,C 180.00000} ; retreat
  ; Step 2850, bar 2896
  LIN {X 374.916,Y -231.794,Z 1086.991,A 92.55766,B 0.00000,C -180.00000} ; outside
  LIN {X 374.916,Y -231.794,Z 121.006,A 92.55766,B 0.00000,C -180.00000} ; preinsert
  LIN {X 374.916,Y -231.794,Z -128.994,A 92.55766,B 0.00000,C -180.00000} ; insert
  LIN {X 374.916,Y -231.794,Z -128.994,A 92.55766,B 0.00000,C -180.00000} ; release
  LIN {X 374.916,Y -231.794,Z 171.006,A 92.55766,B 0.00000,C -180.00000} ; retreat
  ; Step 2851, bar 2898
  LIN {X 1124.916,Y -231.794,Z 1086.991,A 92.55766,B 0.00000,C 180.00000} ; outside
  LIN {X 1124.916,Y -231.794,Z 121.006,A 92.55766,B 0.00000,C 180.00000} ; preinsert
  LIN {X 1124.916,Y -231.794,Z -128.994,A 92.55766,B 0.00000,C 180.00000} ; insert
  LIN {X 1124.916,Y -231.794,Z -128.994,A 92.55766,B 0.00000,C 180.00000} ; release
  LIN {X 1124.916,Y -231.794,Z 171.006,A 92.55766,B 0.00000,C 180.00000} ; retreat
  ; Step 2852, bar 2901
  LIN {X 1874.916,Y -231.794,Z 1086.991,A 92.55766,B 0.00000,C 180.00000} ; outside
  LIN {X 1874.916,Y -231.794,Z 121.006,A 92.55766,B 0.00000,C 180.00000} ; preinsert
  LIN {X 1874.916,Y -231.794,Z -128.994,A 92.55766,B 0.00000,C 180.00000} ; insert
  LIN {X 1874.916,Y -231.794,Z -128.994,A 92.55766,B 0.00000,C 180.00000} ; release
  LIN {X 1874.916,Y -231.794,Z 171.006,A 92.55766,B 0.00000,C 180.00000} ; retreat
  ; Step 2853, bar 2904
  LIN {X 2624.916,Y -231.794,Z 1086.991,A 92.55766,B 0.00000,C 180.00000} ; outside
  LIN {X 2624.916,Y -231.794,Z 121.006,A 92.55766,B 0.00000,C 180.00000} ; preinsert
  LIN {X 2624.916,Y -231.794,Z -128.994,A 92.55766,B 0.00000,C 180.00000} ; insert
  LIN {X 2624.916,Y -231.794,Z -128.994,A 92.55766,B 0.00000,C 180.00000} ; release
  LIN {X 2624.916,Y -231.794,Z 171.006,A 92.55766,B 0.00000,C 180.00000} ; retreat
  ; Step 2854, bar 2907
  LIN {X 3374.916,Y -231.794,Z 1086.991,A 92.55766,B 0.00000,C 180.00000} ; outside
  LIN {X 3374.916,Y -231.794,Z 121.006,A 92.55766,B 0.00000,C 180.00000} ; preinsert
  LIN {X 3374.916,Y -231.794,Z -128.994,A 92.55766,B 0.00000,C 180.00000} ; insert
  LIN {X 3374.916,Y -231.794,Z -128.994,A 92.55766,B 0.00000,C 180.00000} ; release
  LIN {X 3374.916,Y -231.794,Z 171.006,A 92.55766,B 0.00000,C 180.00000} ; retreat
  ; Step 2855, bar 2910
  LIN {X 4124.916,Y -231.794,Z 1086.991,A 92.55766,B 0.00000,C 180.00000} ; outside
  LIN {X 4124.916,Y -231.794,Z 121.006,A 92.55766,B 0.00000,C 180.00000} ; preinsert
  LIN {X 4124.916,Y -231.794,Z -128.994,A 92.55766,B 0.00000,C 180.00000} ; insert
  LIN {X 4124.916,Y -231.794,Z -128.994,A 92.55766,B 0.00000,C 180.00000} ; release
  LIN {X 4124.916,Y -231.794,Z 171.006,A 92.55766,B 0.00000,C 180.00000} ; retreat
  ; Step 2856, bar 2913
  LIN {X 4874.916,Y -231.794,Z 1086.991,A 92.55766,B 0.00000,C 180.00000} ; outside
  LIN {X 4874.916,Y -231.794,Z 121.006,A 92.55766,B 0.00000,C 180.00000} ; preinsert
  LIN {X 4874.916,Y -231.794,Z -128.994,A 92.55766,B 0.00000,C 180.00000} ; insert
  LIN {X 4874.916,Y -231.794,Z -128.994,A 92.55766,B 0.00000,C 180.00000} ; release
  LIN {X 4874.916,Y -231.794,Z 171.006,A 92.55766,B 0.00000,C 180.00000} ; retreat
  ; Step 2857, bar 2916
  LIN {X 5624.916,Y -231.794,Z 1086.991,A 92.55766,B 0.00000,C 180.00000} ; outside
  LIN {X 5624.916,Y -231.794,Z 121.006,A 92.55766,B 0.00000,C 180.00000} ; preinsert
  LIN {X 5624.916,Y -231.794,Z -128.994,A 92.55766,B 0.00000,C 180.00000} ; insert
  LIN {X 5624.916,Y -231.794,Z -128.994,A 92.55766,B 0.00000,C 180.00000} ; release
  LIN {X 5624.916,Y -231.794,Z 171.006,A 92.55766,B 0.00000,C 180.00000} ; retreat
  ; Step 2858, bar 2919
  LIN {X 6374.916,Y -231.794,Z 1086.991,A 92.55766,B 0.00000,C 180.00000} ; outside
  LIN {X 6374.916,Y -231.794,Z 121.006,A 92.55766,B 0.00000,C 180.00000} ; preinsert
  LIN {X 6374.916,Y -231.794,Z -128.994,A 92.55766,B 0.00000,C 180.00000} ; insert
  LIN {X 6374.916,Y -231.794,Z -128.994,A 92.55766,B 0.00000,C 180.00000} ; release
  LIN {X 6374.916,Y -231.794,Z 171.006,A 92.55766,B 0.00000,C 180.00000} ; retreat
  ; Step 2859, bar 2922
  LIN {X 7124.916,Y -231.794,Z 1086.991,A 92.55766,B 0.00000,C 180.00000} ; outside
  LIN {X 7124.916,Y -231.794,Z 121.006,A 92.55766,B 0.00000,C 180.00000} ; preinsert
  LIN {X 7124.916,Y -231.794,Z -128.994,A 92.55766,B 0.00000,C 180.00000} ; insert
  LIN {X 7124.916,Y -231.794,Z -128.994,A 92.55766,B 0.00000,C 180.00000} ; release
  LIN {X 7124.916,Y -231.794,Z 171.006,A 92.55766,B 0.00000,C 180.00000} ; retreat
  ; Step 2860, bar 2925
  LIN {X 7874.916,Y -231.794,Z 1086.991,A 92.55766,B 0.00000,C 180.00000} ; outside
  LIN {X 7874.916,Y -231.794,Z 121.006,A 92.55766,B 0.00000,C 180.00000} ; preinsert
  LIN {X 7874.916,Y -231.794,Z -128.994,A 92.55766,B 0.00000,C 180.00000} ; insert
  LIN {X 7874.916,Y -231.794,Z -128.994,A 92.55766,B 0.00000,C 180.00000} ; release
  LIN {X 7874.916,Y -231.794,Z 171.006,A 92.55766,B 0.00000,C 180.00000} ; retreat
  ; Step 2861, bar 2928
  LIN {X 8624.916,Y -231.794,Z 1086.991,A 92.55766,B 0.00000,C 180.00000} ; outside
  LIN {X 8624.916,Y -231.794,Z 121.006,A 92.55766,B 0.00000,C 180.00000} ; preinsert
  LIN {X 8624.916,Y -231.794,Z -128.994,A 92.55766,B 0.00000,C 180.00000} ; insert
  LIN {X 8624.916,Y -231.794,Z -128.994,A 92.55766,B 0.00000,C 180.00000} ; release
  LIN {X 8624.916,Y -231.794,Z 171.006,A 92.55766,B 0.00000,C 180.00000} ; retreat
  ; Step 2862, bar 2931
  LIN {X 9374.916,Y -231.794,Z 1086.991,A 92.55766,B 0.00000,C 180.00000} ; outside
  LIN {X 9374.916,Y -231.794,Z 121.006,A 92.55766,B 0.00000,C 180.00000} ; preinsert
  LIN {X 9374.916,Y -231.794,Z -128.994,A 92.55766,B 0.00000,C 180.00000} ; insert
  LIN {X 9374.916,Y -231.794,Z -128.994,A 92.55766,B 0.00000,C 180.00000} ; release
  LIN {X 9374.916,Y -231.794,Z 171.006,A 92.55766,B 0.00000,C 180.00000} ; retreat
  ; Step 2863, bar 2934
  LIN {X 10124.916,Y -231.794,Z 1086.991,A 92.55766,B 0.00000,C 180.00000} ; outside
  LIN {X 10124.916,Y -231.794,Z 121.006,A 92.55766,B 0.00000,C 180.00000} ; preinsert
  LIN {X 10124.916,Y -231.794,Z -128.994,A 92.55766,B 0.00000,C 180.00000} ; insert
  LIN {X 10124.916,Y -231.794,Z -128.994,A 92.55766,B 0.00000,C 180.00000} ; release
  LIN {X 10124.916,Y -231.794,Z 171.006,A 92.55766,B 0.00000,C 180.00000} ; retreat
  ; Step 2864, bar 2937
  LIN {X 10874.916,Y -231.794,Z 1086.991,A 92.55766,B 0.00000,C 180.00000} ; outside
  LIN {X 10874.916,Y -231.794,Z 121.006,A 92.55766,B 0.00000,C 180.00000} ; preinsert
  LIN {X 10874.916,Y -231.794,Z -128.994,A 92.55766,B 0.00000,C 180.00000} ; insert
  LIN {X 10874.916,Y -231.794,Z -128.994,A 92.55766,B 0.00000,C 180.00000} ; release
  LIN {X 10874.916,Y -231.794,Z 171.006,A 92.55766,B 0.00000,C 180.00000} ; retreat
  ; Step 2865, bar 2940
  LIN {X 11624.916,Y -231.794,Z 1086.991,A 92.55766,B 0.00000,C 180.00000} ; outside
  LIN {X 11624.916,Y -231.794,Z 121.006,A 92.55766,B 0.00000,C 180.00000} ; preinsert
  LIN {X 11624.916,Y -231.794,Z -128.994,A 92.55766,B 0.00000,C 180.00000} ; insert
  LIN {X 11624.916,Y -231.794,Z -128.994,A 92.55766,B 0.00000,C 180.00000} ; release
  LIN {X 11624.916,Y -231.794,Z 171.006,A 92.55766,B 0.00000,C 180.00000} ; retreat
  ; Step 2866, bar 2630
  LIN {X -11624.916,Y 231.794,Z 1086.991,A -87.44234,B 0.00000,C 180.00000} ; outside
  LIN {X -11624.916,Y 231.794,Z 121.006,A -87.44234,B 0.00000,C 180.00000} ; preinsert
  LIN {X -11624.916,Y 231.794,Z -128.994,A -87.44234,B 0.00000,C 180.00000} ; insert
  LIN {X -11624.916,Y 231.794,Z -128.994,A -87.44234,B 0.00000,C 180.00000} ; release
  LIN {X -11624.916,Y 231.794,Z 171.006,A -87.44234,B 0.00000,C 180.00000} ; retreat
  ; Step 2867, bar 2623
  LIN {X -10874.916,Y 231.794,Z 1086.991,A -87.44234,B 0.00000,C 180.00000} ; outside
  LIN {X -10874.916,Y 231.794,Z 121.006,A -87.44234,B 0.00000,C 180.00000} ; preinsert
  LIN {X -10874.916,Y 231.794,Z -128.994,A -87.44234,B 0.00000,C 180.00000} ; insert
  LIN {X -10874.916,Y 231.794,Z -128.994,A -87.44234,B 0.00000,C 180.00000} ; release
  LIN {X -10874.916,Y 231.794,Z 171.006,A -87.44234,B 0.00000,C 180.00000} ; retreat
  ; Step 2868, bar 2616
  LIN {X -10124.916,Y 231.794,Z 1086.991,A -87.44234,B 0.00000,C 180.00000} ; outside
  LIN {X -10124.916,Y 231.794,Z 121.006,A -87.44234,B 0.00000,C 180.00000} ; preinsert
  LIN {X -10124.916,Y 231.794,Z -128.994,A -87.44234,B 0.00000,C 180.00000} ; insert
  LIN {X -10124.916,Y 231.794,Z -128.994,A -87.44234,B 0.00000,C 180.00000} ; release
  LIN {X -10124.916,Y 231.794,Z 171.006,A -87.44234,B 0.00000,C 180.00000} ; retreat
  ; Step 2869, bar 2609
  LIN {X -9374.916,Y 231.794,Z 1086.991,A -87.44234,B 0.00000,C 180.00000} ; outside
  LIN {X -9374.916,Y 231.794,Z 121.006,A -87.44234,B 0.00000,C 180.00000} ; preinsert
  LIN {X -9374.916,Y 231.794,Z -128.994,A -87.44234,B 0.00000,C 180.00000} ; insert
  LIN {X -9374.916,Y 231.794,Z -128.994,A -87.44234,B 0.00000,C 180.00000} ; release
  LIN {X -9374.916,Y 231.794,Z 171.006,A -87.44234,B 0.00000,C 180.00000} ; retreat
  ; Step 2870, bar 2602
  LIN {X -8624.916,Y 231.794,Z 1086.991,A -87.44234,B 0.00000,C 180.00000} ; outside
  LIN {X -8624.916,Y 231.794,Z 121.006,A -87.44234,B 0.00000,C 180.00000} ; preinsert
  LIN {X -8624.916,Y 231.794,Z -128.994,A -87.44234,B 0.00000,C 180.00000} ; insert
  LIN {X -8624.916,Y 231.794,Z -128.994,A -87.44234,B 0.00000,C 180.00000} ; release
  LIN {X -8624.916,Y 231.794,Z 171.006,A -87.44234,B 0.00000,C 180.00000} ; retreat
  ; Step 2871, bar 2595
  LIN {X -7874.916,Y 231.794,Z 1086.991,A -87.44234,B 0.00000,C 180.00000} ; outside
  LIN {X -7874.916,Y 231.794,Z 121.006,A -87.44234,B 0.00000,C 180.00000} ; preinsert
  LIN {X -7874.916,Y 231.794,Z -128.994,A -87.44234,B 0.00000,C 180.00000} ; insert
  LIN {X -7874.916,Y 231.794,Z -128.994,A -87.44234,B 0.00000,C 180.00000} ; release
  LIN {X -7874.916,Y 231.794,Z 171.006,A -87.44234,B 0.00000,C 180.00000} ; retreat
  ; Step 2872, bar 2588
  LIN {X -7124.916,Y 231.794,Z 1086.991,A -87.44234,B 0.00000,C 180.00000} ; outside
  LIN {X -7124.916,Y 231.794,Z 121.006,A -87.44234,B 0.00000,C 180.00000} ; preinsert
  LIN {X -7124.916,Y 231.794,Z -128.994,A -87.44234,B 0.00000,C 180.00000} ; insert
  LIN {X -7124.916,Y 231.794,Z -128.994,A -87.44234,B 0.00000,C 180.00000} ; release
  LIN {X -7124.916,Y 231.794,Z 171.006,A -87.44234,B 0.00000,C 180.00000} ; retreat
  ; Step 2873, bar 2581
  LIN {X -6374.916,Y 231.794,Z 1086.991,A -87.44234,B 0.00000,C 180.00000} ; outside
  LIN {X -6374.916,Y 231.794,Z 121.006,A -87.44234,B 0.00000,C 180.00000} ; preinsert
  LIN {X -6374.916,Y 231.794,Z -128.994,A -87.44234,B 0.00000,C 180.00000} ; insert
  LIN {X -6374.916,Y 231.794,Z -128.994,A -87.44234,B 0.00000,C 180.00000} ; release
  LIN {X -6374.916,Y 231.794,Z 171.006,A -87.44234,B 0.00000,C 180.00000} ; retreat
  ; Step 2874, bar 2574
  LIN {X -5624.916,Y 231.794,Z 1086.991,A -87.44234,B 0.00000,C 180.00000} ; outside
  LIN {X -5624.916,Y 231.794,Z 121.006,A -87.44234,B 0.00000,C 180.00000} ; preinsert
  LIN {X -5624.916,Y 231.794,Z -128.994,A -87.44234,B 0.00000,C 180.00000} ; insert
  LIN {X -5624.916,Y 231.794,Z -128.994,A -87.44234,B 0.00000,C 180.00000} ; release
  LIN {X -5624.916,Y 231.794,Z 171.006,A -87.44234,B 0.00000,C 180.00000} ; retreat
  ; Step 2875, bar 2567
  LIN {X -4874.916,Y 231.794,Z 1086.991,A -87.44234,B 0.00000,C 180.00000} ; outside
  LIN {X -4874.916,Y 231.794,Z 121.006,A -87.44234,B 0.00000,C 180.00000} ; preinsert
  LIN {X -4874.916,Y 231.794,Z -128.994,A -87.44234,B 0.00000,C 180.00000} ; insert
  LIN {X -4874.916,Y 231.794,Z -128.994,A -87.44234,B 0.00000,C 180.00000} ; release
  LIN {X -4874.916,Y 231.794,Z 171.006,A -87.44234,B 0.00000,C 180.00000} ; retreat
  ; Step 2876, bar 2560
  LIN {X -4124.916,Y 231.794,Z 1086.991,A -87.44234,B 0.00000,C 180.00000} ; outside
  LIN {X -4124.916,Y 231.794,Z 121.006,A -87.44234,B 0.00000,C 180.00000} ; preinsert
  LIN {X -4124.916,Y 231.794,Z -128.994,A -87.44234,B 0.00000,C 180.00000} ; insert
  LIN {X -4124.916,Y 231.794,Z -128.994,A -87.44234,B 0.00000,C 180.00000} ; release
  LIN {X -4124.916,Y 231.794,Z 171.006,A -87.44234,B 0.00000,C 180.00000} ; retreat
  ; Step 2877, bar 2553
  LIN {X -3374.916,Y 231.794,Z 1086.991,A -87.44234,B 0.00000,C 180.00000} ; outside
  LIN {X -3374.916,Y 231.794,Z 121.006,A -87.44234,B 0.00000,C 180.00000} ; preinsert
  LIN {X -3374.916,Y 231.794,Z -128.994,A -87.44234,B 0.00000,C 180.00000} ; insert
  LIN {X -3374.916,Y 231.794,Z -128.994,A -87.44234,B 0.00000,C 180.00000} ; release
  LIN {X -3374.916,Y 231.794,Z 171.006,A -87.44234,B 0.00000,C 180.00000} ; retreat
  ; Step 2878, bar 2546
  LIN {X -2624.916,Y 231.794,Z 1086.991,A -87.44234,B 0.00000,C 180.00000} ; outside
  LIN {X -2624.916,Y 231.794,Z 121.006,A -87.44234,B 0.00000,C 180.00000} ; preinsert
  LIN {X -2624.916,Y 231.794,Z -128.994,A -87.44234,B 0.00000,C 180.00000} ; insert
  LIN {X -2624.916,Y 231.794,Z -128.994,A -87.44234,B 0.00000,C 180.00000} ; release
  LIN {X -2624.916,Y 231.794,Z 171.006,A -87.44234,B 0.00000,C 180.00000} ; retreat
  ; Step 2879, bar 2539
  LIN {X -1874.916,Y 231.794,Z 1086.991,A -87.44234,B 0.00000,C 180.00000} ; outside
  LIN {X -1874.916,Y 231.794,Z 121.006,A -87.44234,B 0.00000,C 180.00000} ; preinsert
  LIN {X -1874.916,Y 231.794,Z -128.994,A -87.44234,B 0.00000,C 180.00000} ; insert
  LIN {X -1874.916,Y 231.794,Z -128.994,A -87.44234,B 0.00000,C 180.00000} ; release
  LIN {X -1874.916,Y 231.794,Z 171.006,A -87.44234,B 0.00000,C 180.00000} ; retreat
  ; Step 2880, bar 2532
  LIN {X -1124.916,Y 231.794,Z 1086.991,A -87.44234,B 0.00000,C 180.00000} ; outside
  LIN {X -1124.916,Y 231.794,Z 121.006,A -87.44234,B 0.00000,C 180.00000} ; preinsert
  LIN {X -1124.916,Y 231.794,Z -128.994,A -87.44234,B 0.00000,C 180.00000} ; insert
  LIN {X -1124.916,Y 231.794,Z -128.994,A -87.44234,B 0.00000,C 180.00000} ; release
  LIN {X -1124.916,Y 231.794,Z 171.006,A -87.44234,B 0.00000,C 180.00000} ; retreat
  ; Step 2881, bar 1973
  LIN {X -374.916,Y 231.794,Z 1086.991,A -87.44234,B 0.00000,C 180.00000} ; outside
  LIN {X -374.916,Y 231.794,Z 121.006,A -87.44234,B 0.00000,C 180.00000} ; preinsert
  LIN {X -374.916,Y 231.794,Z -128.994,A -87.44234,B 0.00000,C 180.00000} ; insert
  LIN {X -374.916,Y 231.794,Z -128.994,A -87.44234,B 0.00000,C 180.00000} ; release
  LIN {X -374.916,Y 231.794,Z 171.006,A -87.44234,B 0.00000,C 180.00000} ; retreat
  ; Step 2882, bar 2685
  LIN {X 374.916,Y 231.794,Z 1086.991,A -92.55766,B 0.00000,C 180.00000} ; outside
  LIN {X 374.916,Y 231.794,Z 121.006,A -92.55766,B 0.00000,C 180.00000} ; preinsert
  LIN {X 374.916,Y 231.794,Z -128.994,A -92.55766,B 0.00000,C 180.00000} ; insert
  LIN {X 374.916,Y 231.794,Z -128.994,A -92.55766,B 0.00000,C 180.00000} ; release
  LIN {X 374.916,Y 231.794,Z 171.006,A -92.55766,B 0.00000,C 180.00000} ; retreat
  ; Step 2883, bar 2688
  LIN {X 1124.916,Y 231.794,Z 1086.991,A -92.55766,B 0.00000,C -180.00000} ; outside
  LIN {X 1124.916,Y 231.794,Z 121.006,A -92.55766,B 0.00000,C -180.00000} ; preinsert
  LIN {X 1124.916,Y 231.794,Z -128.994,A -92.55766,B 0.00000,C -180.00000} ; insert
  LIN {X 1124.916,Y 231.794,Z -128.994,A -92.55766,B 0.00000,C -180.00000} ; release
  LIN {X 1124.916,Y 231.794,Z 171.006,A -92.55766,B 0.00000,C -180.00000} ; retreat
  ; Step 2884, bar 2692
  LIN {X 1874.916,Y 231.794,Z 1086.991,A -92.55766,B 0.00000,C -180.00000} ; outside
  LIN {X 1874.916,Y 231.794,Z 121.006,A -92.55766,B 0.00000,C -180.00000} ; preinsert
  LIN {X 1874.916,Y 231.794,Z -128.994,A -92.55766,B 0.00000,C -180.00000} ; insert
  LIN {X 1874.916,Y 231.794,Z -128.994,A -92.55766,B 0.00000,C -180.00000} ; release
  LIN {X 1874.916,Y 231.794,Z 171.006,A -92.55766,B 0.00000,C -180.00000} ; retreat
  ; Step 2885, bar 2696
  LIN {X 2624.916,Y 231.794,Z 1086.991,A -92.55766,B 0.00000,C -180.00000} ; outside
  LIN {X 2624.916,Y 231.794,Z 121.006,A -92.55766,B 0.00000,C -180.00000} ; preinsert
  LIN {X 2624.916,Y 231.794,Z -128.994,A -92.55766,B 0.00000,C -180.00000} ; insert
  LIN {X 2624.916,Y 231.794,Z -128.994,A -92.55766,B 0.00000,C -180.00000} ; release
  LIN {X 2624.916,Y 231.794,Z 171.006,A -92.55766,B 0.00000,C -180.00000} ; retreat
  ; Step 2886, bar 2700
  LIN {X 3374.916,Y 231.794,Z 1086.991,A -92.55766,B 0.00000,C -180.00000} ; outside
  LIN {X 3374.916,Y 231.794,Z 121.006,A -92.55766,B 0.00000,C -180.00000} ; preinsert
  LIN {X 3374.916,Y 231.794,Z -128.994,A -92.55766,B 0.00000,C -180.00000} ; insert
  LIN {X 3374.916,Y 231.794,Z -128.994,A -92.55766,B 0.00000,C -180.00000} ; release
  LIN {X 3374.916,Y 231.794,Z 171.006,A -92.55766,B 0.00000,C -180.00000} ; retreat
  ; Step 2887, bar 2704
  LIN {X 4124.916,Y 231.794,Z 1086.991,A -92.55766,B 0.00000,C -180.00000} ; outside
  LIN {X 4124.916,Y 231.794,Z 121.006,A -92.55766,B 0.00000,C -180.00000} ; preinsert
  LIN {X 4124.916,Y 231.794,Z -128.994,A -92.55766,B 0.00000,C -180.00000} ; insert
  LIN {X 4124.916,Y 231.794,Z -128.994,A -92.55766,B 0.00000,C -180.00000} ; release
  LIN {X 4124.916,Y 231.794,Z 171.006,A -92.55766,B 0.00000,C -180.00000} ; retreat
  ; Step 2888, bar 2708
  LIN {X 4874.916,Y 231.794,Z 1086.991,A -92.55766,B 0.00000,C -180.00000} ; outside
  LIN {X 4874.916,Y 231.794,Z 121.006,A -92.55766,B 0.00000,C -180.00000} ; preinsert
  LIN {X 4874.916,Y 231.794,Z -128.994,A -92.55766,B 0.00000,C -180.00000} ; insert
  LIN {X 4874.916,Y 231.794,Z -128.994,A -92.55766,B 0.00000,C -180.00000} ; release
  LIN {X 4874.916,Y 231.794,Z 171.006,A -92.55766,B 0.00000,C -180.00000} ; retreat
  ; Step 2889, bar 2712
  LIN {X 5624.916,Y 231.794,Z 1086.991,A -92.55766,B 0.00000,C -180.00000} ; outside
  LIN {X 5624.916,Y 231.794,Z 121.006,A -92.55766,B 0.00000,C -180.00000} ; preinsert
  LIN {X 5624.916,Y 231.794,Z -128.994,A -92.55766,B 0.00000,C -180.00000} ; insert
  LIN {X 5624.916,Y 231.794,Z -128.994,A -92.55766,B 0.00000,C -180.00000} ; release
  LIN {X 5624.916,Y 231.794,Z 171.006,A -92.55766,B 0.00000,C -180.00000} ; retreat
  ; Step 2890, bar 2716
  LIN {X 6374.916,Y 231.794,Z 1086.991,A -92.55766,B 0.00000,C -180.00000} ; outside
  LIN {X 6374.916,Y 231.794,Z 121.006,A -92.55766,B 0.00000,C -180.00000} ; preinsert
  LIN {X 6374.916,Y 231.794,Z -128.994,A -92.55766,B 0.00000,C -180.00000} ; insert
  LIN {X 6374.916,Y 231.794,Z -128.994,A -92.55766,B 0.00000,C -180.00000} ; release
  LIN {X 6374.916,Y 231.794,Z 171.006,A -92.55766,B 0.00000,C -180.00000} ; retreat
  ; Step 2891, bar 2720
  LIN {X 7124.916,Y 231.794,Z 1086.991,A -92.55766,B 0.00000,C -180.00000} ; outside
  LIN {X 7124.916,Y 231.794,Z 121.006,A -92.55766,B 0.00000,C -180.00000} ; preinsert
  LIN {X 7124.916,Y 231.794,Z -128.994,A -92.55766,B 0.00000,C -180.00000} ; insert
  LIN {X 7124.916,Y 231.794,Z -128.994,A -92.55766,B 0.00000,C -180.00000} ; release
  LIN {X 7124.916,Y 231.794,Z 171.006,A -92.55766,B 0.00000,C -180.00000} ; retreat
  ; Step 2892, bar 2724
  LIN {X 7874.916,Y 231.794,Z 1086.991,A -92.55766,B 0.00000,C -180.00000} ; outside
  LIN {X 7874.916,Y 231.794,Z 121.006,A -92.55766,B 0.00000,C -180.00000} ; preinsert
  LIN {X 7874.916,Y 231.794,Z -128.994,A -92.55766,B 0.00000,C -180.00000} ; insert
  LIN {X 7874.916,Y 231.794,Z -128.994,A -92.55766,B 0.00000,C -180.00000} ; release
  LIN {X 7874.916,Y 231.794,Z 171.006,A -92.55766,B 0.00000,C -180.00000} ; retreat
  ; Step 2893, bar 2728
  LIN {X 8624.916,Y 231.794,Z 1086.991,A -92.55766,B 0.00000,C -180.00000} ; outside
  LIN {X 8624.916,Y 231.794,Z 121.006,A -92.55766,B 0.00000,C -180.00000} ; preinsert
  LIN {X 8624.916,Y 231.794,Z -128.994,A -92.55766,B 0.00000,C -180.00000} ; insert
  LIN {X 8624.916,Y 231.794,Z -128.994,A -92.55766,B 0.00000,C -180.00000} ; release
  LIN {X 8624.916,Y 231.794,Z 171.006,A -92.55766,B 0.00000,C -180.00000} ; retreat
  ; Step 2894, bar 2732
  LIN {X 9374.916,Y 231.794,Z 1086.991,A -92.55766,B 0.00000,C -180.00000} ; outside
  LIN {X 9374.916,Y 231.794,Z 121.006,A -92.55766,B 0.00000,C -180.00000} ; preinsert
  LIN {X 9374.916,Y 231.794,Z -128.994,A -92.55766,B 0.00000,C -180.00000} ; insert
  LIN {X 9374.916,Y 231.794,Z -128.994,A -92.55766,B 0.00000,C -180.00000} ; release
  LIN {X 9374.916,Y 231.794,Z 171.006,A -92.55766,B 0.00000,C -180.00000} ; retreat
  ; Step 2895, bar 2736
  LIN {X 10124.916,Y 231.794,Z 1086.991,A -92.55766,B 0.00000,C -180.00000} ; outside
  LIN {X 10124.916,Y 231.794,Z 121.006,A -92.55766,B 0.00000,C -180.00000} ; preinsert
  LIN {X 10124.916,Y 231.794,Z -128.994,A -92.55766,B 0.00000,C -180.00000} ; insert
  LIN {X 10124.916,Y 231.794,Z -128.994,A -92.55766,B 0.00000,C -180.00000} ; release
  LIN {X 10124.916,Y 231.794,Z 171.006,A -92.55766,B 0.00000,C -180.00000} ; retreat
  ; Step 2896, bar 2740
  LIN {X 10874.916,Y 231.794,Z 1086.991,A -92.55766,B 0.00000,C -180.00000} ; outside
  LIN {X 10874.916,Y 231.794,Z 121.006,A -92.55766,B 0.00000,C -180.00000} ; preinsert
  LIN {X 10874.916,Y 231.794,Z -128.994,A -92.55766,B 0.00000,C -180.00000} ; insert
  LIN {X 10874.916,Y 231.794,Z -128.994,A -92.55766,B 0.00000,C -180.00000} ; release
  LIN {X 10874.916,Y 231.794,Z 171.006,A -92.55766,B 0.00000,C -180.00000} ; retreat
  ; Step 2897, bar 2744
  LIN {X 11624.916,Y 231.794,Z 1086.991,A -92.55766,B 0.00000,C -180.00000} ; outside
  LIN {X 11624.916,Y 231.794,Z 121.006,A -92.55766,B 0.00000,C -180.00000} ; preinsert
  LIN {X 11624.916,Y 231.794,Z -128.994,A -92.55766,B 0.00000,C -180.00000} ; insert
  LIN {X 11624.916,Y 231.794,Z -128.994,A -92.55766,B 0.00000,C -180.00000} ; release
  LIN {X 11624.916,Y 231.794,Z 171.006,A -92.55766,B 0.00000,C -180.00000} ; retreat
  ; Step 2898, bar 1857
  LIN {X -14549.934,Y -0.335,Z 839.906,A 89.99422,B 0.00000,C -180.00000} ; outside
  LIN {X -14549.934,Y -0.335,Z -123.558,A 89.99422,B 0.00000,C -180.00000} ; preinsert
  LIN {X -14549.934,Y -0.335,Z -373.558,A 89.99422,B 0.00000,C -180.00000} ; insert
  LIN {X -14549.934,Y -0.335,Z -373.558,A 89.99422,B 0.00000,C -180.00000} ; release
  LIN {X -14549.934,Y -0.335,Z -73.558,A 89.99422,B 0.00000,C -180.00000} ; retreat
  ; Step 2899, bar 1044
  LIN {X 14549.934,Y -0.335,Z 839.906,A 90.00578,B 0.00000,C 180.00000} ; outside
  LIN {X 14549.934,Y -0.335,Z -123.558,A 90.00578,B 0.00000,C 180.00000} ; preinsert
  LIN {X 14549.934,Y -0.335,Z -373.558,A 90.00578,B 0.00000,C 180.00000} ; insert
  LIN {X 14549.934,Y -0.335,Z -373.558,A 90.00578,B 0.00000,C 180.00000} ; release
  LIN {X 14549.934,Y -0.335,Z -73.558,A 90.00578,B 0.00000,C 180.00000} ; retreat
  ; Step 2900, bar 3048
  LIN {X -15849.996,Y -231.529,Z 999.648,A -172.46345,B 0.00000,C 180.00000} ; outside
  LIN {X -15849.996,Y -231.529,Z 30.709,A -172.46345,B 0.00000,C 180.00000} ; preinsert
  LIN {X -15849.996,Y -231.529,Z -219.291,A -172.46345,B 0.00000,C 180.00000} ; insert
  LIN {X -15849.996,Y -231.529,Z -219.291,A -172.46345,B 0.00000,C 180.00000} ; release
  LIN {X -15849.996,Y -231.529,Z 80.709,A -172.46345,B 0.00000,C 180.00000} ; retreat
  ; Step 2901, bar 3043
  LIN {X -15449.996,Y -231.529,Z 999.648,A -172.46345,B 0.00000,C 180.00000} ; outside
  LIN {X -15449.996,Y -231.529,Z 30.709,A -172.46345,B 0.00000,C 180.00000} ; preinsert
  LIN {X -15449.996,Y -231.529,Z -219.291,A -172.46345,B 0.00000,C 180.00000} ; insert
  LIN {X -15449.996,Y -231.529,Z -219.291,A -172.46345,B 0.00000,C 180.00000} ; release
  LIN {X -15449.996,Y -231.529,Z 80.709,A -172.46345,B 0.00000,C 180.00000} ; retreat
  ; Step 2902, bar 3076
  LIN {X 15449.996,Y -231.529,Z 999.647,A -7.53655,B 0.00000,C 180.00000} ; outside
  LIN {X 15449.996,Y -231.529,Z 30.709,A -7.53655,B 0.00000,C 180.00000} ; preinsert
  LIN {X 15449.996,Y -231.529,Z -219.291,A -7.53655,B 0.00000,C 180.00000} ; insert
  LIN {X 15449.996,Y -231.529,Z -219.291,A -7.53655,B 0.00000,C 180.00000} ; release
  LIN {X 15449.996,Y -231.529,Z 80.709,A -7.53655,B 0.00000,C 180.00000} ; retreat
  ; Step 2903, bar 3081
  LIN {X 15849.996,Y -231.529,Z 999.647,A -7.53655,B 0.00000,C 180.00000} ; outside
  LIN {X 15849.996,Y -231.529,Z 30.709,A -7.53655,B 0.00000,C 180.00000} ; preinsert
  LIN {X 15849.996,Y -231.529,Z -219.291,A -7.53655,B 0.00000,C 180.00000} ; insert
  LIN {X 15849.996,Y -231.529,Z -219.291,A -7.53655,B 0.00000,C 180.00000} ; release
  LIN {X 15849.996,Y -231.529,Z 80.709,A -7.53655,B 0.00000,C 180.00000} ; retreat
  ; Step 2904, bar 3053
  LIN {X -16249.996,Y -231.529,Z 999.648,A -172.46345,B 0.00000,C 180.00000} ; outside
  LIN {X -16249.996,Y -231.529,Z 30.709,A -172.46345,B 0.00000,C 180.00000} ; preinsert
  LIN {X -16249.996,Y -231.529,Z -219.291,A -172.46345,B 0.00000,C 180.00000} ; insert
  LIN {X -16249.996,Y -231.529,Z -219.291,A -172.46345,B 0.00000,C 180.00000} ; release
  LIN {X -16249.996,Y -231.529,Z 80.709,A -172.46345,B 0.00000,C 180.00000} ; retreat
  ; Step 2905, bar 3086
  LIN {X 16249.996,Y -231.529,Z 999.647,A -7.53655,B 0.00000,C 180.00000} ; outside
  LIN {X 16249.996,Y -231.529,Z 30.709,A -7.53655,B 0.00000,C 180.00000} ; preinsert
  LIN {X 16249.996,Y -231.529,Z -219.291,A -7.53655,B 0.00000,C 180.00000} ; insert
  LIN {X 16249.996,Y -231.529,Z -219.291,A -7.53655,B 0.00000,C 180.00000} ; release
  LIN {X 16249.996,Y -231.529,Z 80.709,A -7.53655,B 0.00000,C 180.00000} ; retreat
  ; Step 2906, bar 3038
  LIN {X -16249.996,Y 231.529,Z 999.647,A 172.46345,B 0.00000,C -180.00000} ; outside
  LIN {X -16249.996,Y 231.529,Z 30.709,A 172.46345,B 0.00000,C -180.00000} ; preinsert
  LIN {X -16249.996,Y 231.529,Z -219.291,A 172.46345,B 0.00000,C -180.00000} ; insert
  LIN {X -16249.996,Y 231.529,Z -219.291,A 172.46345,B 0.00000,C -180.00000} ; release
  LIN {X -16249.996,Y 231.529,Z 80.709,A 172.46345,B 0.00000,C -180.00000} ; retreat
  ; Step 2907, bar 3032
  LIN {X -15849.996,Y 231.529,Z 999.647,A 172.46345,B 0.00000,C -180.00000} ; outside
  LIN {X -15849.996,Y 231.529,Z 30.709,A 172.46345,B 0.00000,C -180.00000} ; preinsert
  LIN {X -15849.996,Y 231.529,Z -219.291,A 172.46345,B 0.00000,C -180.00000} ; insert
  LIN {X -15849.996,Y 231.529,Z -219.291,A 172.46345,B 0.00000,C -180.00000} ; release
